   DATA[2577,13] := 828.5936;
   DATA[2577,14] := 1.0;
   DATA[2577,15] := 2.0;
   DATA[2577,16] := 1.0;
   DATA[2577,17] := 1.0;
   DATA[2577,18] := 1.0;
   DATA[2577,19] := 2.0;
   DATA[2577,20] := 148.808;
   DATA[2577,21] := 155.191;
   DATA[2577,22] := 1.713261;
   DATA[2577,23] := 874.6988;
   DATA[2577,24] := 2.0;
   DATA[2577,25] := 2.0;
   DATA[2577,26] := 7.871251;
   DATA[2577,27] := 144.4758;
   DATA[2577,28] := 261.3753;
   DATA[2577,29] := 12.03538;
   DATA[2577,30] := 1.724301;
   DATA[2577,31] := 1.29243;
   DATA[2577,32] := 0.7352687;
   DATA[2577,33] := 0.3084265;
   DATA[2577,34] := 2.0;
   DATA[2577,35] := 249.6155;
   DATA[2577,36] := 1.649953;
   DATA[2577,37] := 188.5254;
   DATA[2577,38] := 0.000128152;
   DATA[2577,39] := 1.0;
   DATA[2577,40] := 1.0;
   DATA[2578,0] := 2.550043;
   DATA[2578,1] := 868.9383;
   DATA[2578,2] := 2.0;
   DATA[2578,3] := 2.0;
   DATA[2578,4] := 262.3366;
   DATA[2578,5] := 8.396437;
   DATA[2578,6] := 329.4027;
   DATA[2578,7] := 2.452312;
   DATA[2578,8] := 2.0;
   DATA[2578,9] := 2.0;
   DATA[2578,10] := 2.0;
   DATA[2578,11] := 19.68756;
   DATA[2578,12] := 2.209653;
   DATA[2578,13] := 829.0342;
   DATA[2578,14] := 1.0;
   DATA[2578,15] := 2.0;
   DATA[2578,16] := 1.0;
   DATA[2578,17] := 1.0;
   DATA[2578,18] := 1.0;
   DATA[2578,19] := 2.0;
   DATA[2578,20] := 148.808;
   DATA[2578,21] := 155.191;
   DATA[2578,22] := 1.713261;
   DATA[2578,23] := 874.8141;
   DATA[2578,24] := 2.0;
   DATA[2578,25] := 2.0;
   DATA[2578,26] := 7.872853;
   DATA[2578,27] := 144.4758;
   DATA[2578,28] := 261.3753;
   DATA[2578,29] := 12.03538;
   DATA[2578,30] := 1.724301;
   DATA[2578,31] := 1.301524;
   DATA[2578,32] := 0.7352687;
   DATA[2578,33] := 0.3084265;
   DATA[2578,34] := 2.0;
   DATA[2578,35] := 249.8718;
   DATA[2578,36] := 1.649953;
   DATA[2578,37] := 188.7176;
   DATA[2578,38] := 0.000128152;
   DATA[2578,39] := 1.0;
   DATA[2578,40] := 1.0;
   DATA[2579,0] := 2.586875;
   DATA[2579,1] := 868.5458;
   DATA[2579,2] := 2.0;
   DATA[2579,3] := 2.0;
   DATA[2579,4] := 262.3366;
   DATA[2579,5] := 8.396437;
   DATA[2579,6] := 329.4027;
   DATA[2579,7] := 2.451927;
   DATA[2579,8] := 2.0;
   DATA[2579,9] := 2.0;
   DATA[2579,10] := 2.0;
   DATA[2579,11] := 19.71957;
   DATA[2579,12] := 2.209653;
   DATA[2579,13] := 829.3547;
   DATA[2579,14] := 1.0;
   DATA[2579,15] := 2.0;
   DATA[2579,16] := 1.0;
   DATA[2579,17] := 1.0;
   DATA[2579,18] := 1.0;
   DATA[2579,19] := 2.0;
   DATA[2579,20] := 148.808;
   DATA[2579,21] := 155.191;
   DATA[2579,22] := 1.716208;
   DATA[2579,23] := 875.0064;
   DATA[2579,24] := 2.0;
   DATA[2579,25] := 2.0;
   DATA[2579,26] := 7.872853;
   DATA[2579,27] := 144.4758;
   DATA[2579,28] := 261.3753;
   DATA[2579,29] := 12.03538;
   DATA[2579,30] := 1.724686;
   DATA[2579,31] := 1.296657;
   DATA[2579,32] := 0.7352687;
   DATA[2579,33] := 0.3084265;
   DATA[2579,34] := 2.0;
   DATA[2579,35] := 249.8718;
   DATA[2579,36] := 1.649953;
   DATA[2579,37] := 188.7176;
   DATA[2579,38] := 0.000128152;
   DATA[2579,39] := 1.0;
   DATA[2579,40] := 1.0;
   DATA[2580,0] := 2.632995;
   DATA[2580,1] := 868.5458;
   DATA[2580,2] := 2.0;
   DATA[2580,3] := 2.0;
   DATA[2580,4] := 262.3366;
   DATA[2580,5] := 8.396437;
   DATA[2580,6] := 329.4027;
   DATA[2580,7] := 2.451927;
   DATA[2580,8] := 2.0;
   DATA[2580,9] := 2.0;
   DATA[2580,10] := 2.0;
   DATA[2580,11] := 19.74198;
   DATA[2580,12] := 2.208116;
   DATA[2580,13] := 830.4762;
   DATA[2580,14] := 1.0;
   DATA[2580,15] := 2.0;
   DATA[2580,16] := 1.0;
   DATA[2580,17] := 1.0;
   DATA[2580,18] := 1.0;
   DATA[2580,19] := 2.0;
   DATA[2580,20] := 148.808;
   DATA[2580,21] := 155.191;
   DATA[2580,22] := 1.716208;
   DATA[2580,23] := 875.314;
   DATA[2580,24] := 2.0;
   DATA[2580,25] := 2.0;
   DATA[2580,26] := 7.872853;
   DATA[2580,27] := 144.4758;
   DATA[2580,28] := 261.3753;
   DATA[2580,29] := 12.03538;
   DATA[2580,30] := 1.725711;
   DATA[2580,31] := 1.298578;
   DATA[2580,32] := 0.7352687;
   DATA[2580,33] := 0.3084265;
   DATA[2580,34] := 2.0;
   DATA[2580,35] := 249.8718;
   DATA[2580,36] := 1.665972;
   DATA[2580,37] := 188.7176;
   DATA[2580,38] := 0.000128152;
   DATA[2580,39] := 1.0;
   DATA[2580,40] := 1.0;
   DATA[2581,0] := 2.65061;
   DATA[2581,1] := 868.5458;
   DATA[2581,2] := 2.0;
   DATA[2581,3] := 2.0;
   DATA[2581,4] := 262.3366;
   DATA[2581,5] := 8.396437;
   DATA[2581,6] := 329.4027;
   DATA[2581,7] := 2.451927;
   DATA[2581,8] := 2.0;
   DATA[2581,9] := 2.0;
   DATA[2581,10] := 2.0;
   DATA[2581,11] := 19.76439;
   DATA[2581,12] := 2.208116;
   DATA[2581,13] := 830.8767;
   DATA[2581,14] := 1.0;
   DATA[2581,15] := 2.0;
   DATA[2581,16] := 1.0;
   DATA[2581,17] := 1.0;
   DATA[2581,18] := 1.0;
   DATA[2581,19] := 2.0;
   DATA[2581,20] := 148.808;
   DATA[2581,21] := 155.191;
   DATA[2581,22] := 1.716208;
   DATA[2581,23] := 875.3909;
   DATA[2581,24] := 2.0;
   DATA[2581,25] := 2.0;
   DATA[2581,26] := 7.874776;
   DATA[2581,27] := 144.4758;
   DATA[2581,28] := 261.3753;
   DATA[2581,29] := 12.03538;
   DATA[2581,30] := 1.725711;
   DATA[2581,31] := 1.302165;
   DATA[2581,32] := 0.7352687;
   DATA[2581,33] := 0.3084265;
   DATA[2581,34] := 2.0;
   DATA[2581,35] := 249.8718;
   DATA[2581,36] := 1.665972;
   DATA[2581,37] := 188.7176;
   DATA[2581,38] := 0.000128152;
   DATA[2581,39] := 1.0;
   DATA[2581,40] := 1.0;
   DATA[2582,0] := 2.66246;
   DATA[2582,1] := 868.3495;
   DATA[2582,2] := 2.0;
   DATA[2582,3] := 2.0;
   DATA[2582,4] := 262.3366;
   DATA[2582,5] := 8.396437;
   DATA[2582,6] := 329.4027;
   DATA[2582,7] := 2.451927;
   DATA[2582,8] := 2.0;
   DATA[2582,9] := 2.0;
   DATA[2582,10] := 2.0;
   DATA[2582,11] := 19.77079;
   DATA[2582,12] := 2.208116;
   DATA[2582,13] := 831.1971;
   DATA[2582,14] := 1.0;
   DATA[2582,15] := 2.0;
   DATA[2582,16] := 1.0;
   DATA[2582,17] := 1.0;
   DATA[2582,18] := 1.0;
   DATA[2582,19] := 2.0;
   DATA[2582,20] := 148.808;
   DATA[2582,21] := 155.191;
   DATA[2582,22] := 1.716208;
   DATA[2582,23] := 875.3909;
   DATA[2582,24] := 2.0;
   DATA[2582,25] := 2.0;
   DATA[2582,26] := 7.874776;
   DATA[2582,27] := 144.4758;
   DATA[2582,28] := 261.3753;
   DATA[2582,29] := 12.03538;
   DATA[2582,30] := 1.725711;
   DATA[2582,31] := 1.296657;
   DATA[2582,32] := 0.7352687;
   DATA[2582,33] := 0.3084265;
   DATA[2582,34] := 2.0;
   DATA[2582,35] := 249.8718;
   DATA[2582,36] := 1.665972;
   DATA[2582,37] := 188.7176;
   DATA[2582,38] := 0.000128152;
   DATA[2582,39] := 1.0;
   DATA[2582,40] := 1.0;
   DATA[2583,0] := 2.666624;
   DATA[2583,1] := 868.4673;
   DATA[2583,2] := 2.0;
   DATA[2583,3] := 2.0;
   DATA[2583,4] := 262.3366;
   DATA[2583,5] := 8.396437;
   DATA[2583,6] := 329.4027;
   DATA[2583,7] := 2.451927;
   DATA[2583,8] := 2.0;
   DATA[2583,9] := 2.0;
   DATA[2583,10] := 2.0;
   DATA[2583,11] := 19.77079;
   DATA[2583,12] := 2.208116;
   DATA[2583,13] := 831.1971;
   DATA[2583,14] := 1.0;
   DATA[2583,15] := 2.0;
   DATA[2583,16] := 1.0;
   DATA[2583,17] := 1.0;
   DATA[2583,18] := 1.0;
   DATA[2583,19] := 2.0;
   DATA[2583,20] := 148.808;
   DATA[2583,21] := 155.3448;
   DATA[2583,22] := 1.716208;
   DATA[2583,23] := 876.0831;
   DATA[2583,24] := 2.0;
   DATA[2583,25] := 2.0;
   DATA[2583,26] := 7.874776;
   DATA[2583,27] := 144.4758;
   DATA[2583,28] := 261.3753;
   DATA[2583,29] := 12.03538;
   DATA[2583,30] := 1.725711;
   DATA[2583,31] := 1.291277;
   DATA[2583,32] := 0.7352687;
   DATA[2583,33] := 0.3084265;
   DATA[2583,34] := 2.0;
   DATA[2583,35] := 249.8718;
   DATA[2583,36] := 1.665972;
   DATA[2583,37] := 188.7176;
   DATA[2583,38] := 0.000128152;
   DATA[2583,39] := 1.0;
   DATA[2583,40] := 1.0;
   DATA[2584,0] := 2.63844;
   DATA[2584,1] := 868.114;
   DATA[2584,2] := 2.0;
   DATA[2584,3] := 2.0;
   DATA[2584,4] := 262.3366;
   DATA[2584,5] := 8.396437;
   DATA[2584,6] := 329.4027;
   DATA[2584,7] := 2.453209;
   DATA[2584,8] := 2.0;
   DATA[2584,9] := 2.0;
   DATA[2584,10] := 2.0;
   DATA[2584,11] := 19.71637;
   DATA[2584,12] := 2.208116;
   DATA[2584,13] := 831.3574;
   DATA[2584,14] := 1.0;
   DATA[2584,15] := 2.0;
   DATA[2584,16] := 1.0;
   DATA[2584,17] := 1.0;
   DATA[2584,18] := 1.0;
   DATA[2584,19] := 2.0;
   DATA[2584,20] := 148.808;
   DATA[2584,21] := 155.3448;
   DATA[2584,22] := 1.717746;
   DATA[2584,23] := 876.6983;
   DATA[2584,24] := 2.0;
   DATA[2584,25] := 2.0;
   DATA[2584,26] := 7.874776;
   DATA[2584,27] := 144.4758;
   DATA[2584,28] := 261.3753;
   DATA[2584,29] := 12.03538;
   DATA[2584,30] := 1.725711;
   DATA[2584,31] := 1.281286;
   DATA[2584,32] := 0.7352687;
   DATA[2584,33] := 0.3084265;
   DATA[2584,34] := 2.0;
   DATA[2584,35] := 249.9519;
   DATA[2584,36] := 1.665972;
   DATA[2584,37] := 188.7176;
   DATA[2584,38] := 0.000128152;
   DATA[2584,39] := 1.0;
   DATA[2584,40] := 1.0;
   DATA[2585,0] := 2.625308;
   DATA[2585,1] := 868.1533;
   DATA[2585,2] := 2.0;
   DATA[2585,3] := 2.0;
   DATA[2585,4] := 262.3366;
   DATA[2585,5] := 8.396437;
   DATA[2585,6] := 329.4027;
   DATA[2585,7] := 2.453849;
   DATA[2585,8] := 2.0;
   DATA[2585,9] := 2.0;
   DATA[2585,10] := 2.0;
   DATA[2585,11] := 19.68436;
   DATA[2585,12] := 2.208116;
   DATA[2585,13] := 831.1571;
   DATA[2585,14] := 1.0;
   DATA[2585,15] := 2.0;
   DATA[2585,16] := 1.0;
   DATA[2585,17] := 1.0;
   DATA[2585,18] := 1.0;
   DATA[2585,19] := 2.0;
   DATA[2585,20] := 148.808;
   DATA[2585,21] := 155.3448;
   DATA[2585,22] := 1.717746;
   DATA[2585,23] := 876.8521;
   DATA[2585,24] := 2.0;
   DATA[2585,25] := 2.0;
   DATA[2585,26] := 7.874776;
   DATA[2585,27] := 144.4758;
   DATA[2585,28] := 261.3753;
   DATA[2585,29] := 12.03538;
   DATA[2585,30] := 1.726737;
   DATA[2585,31] := 1.281286;
   DATA[2585,32] := 0.7352687;
   DATA[2585,33] := 0.3084265;
   DATA[2585,34] := 2.0;
   DATA[2585,35] := 250.016;
   DATA[2585,36] := 1.665972;
   DATA[2585,37] := 188.7176;
   DATA[2585,38] := 0.000128152;
   DATA[2585,39] := 1.0;
   DATA[2585,40] := 1.0;
   DATA[2586,0] := 2.611536;
   DATA[2586,1] := 867.7607;
   DATA[2586,2] := 2.0;
   DATA[2586,3] := 2.0;
   DATA[2586,4] := 262.3366;
   DATA[2586,5] := 8.396437;
   DATA[2586,6] := 329.4027;
   DATA[2586,7] := 2.455515;
   DATA[2586,8] := 2.0;
   DATA[2586,9] := 2.0;
   DATA[2586,10] := 2.0;
   DATA[2586,11] := 19.68436;
   DATA[2586,12] := 2.208116;
   DATA[2586,13] := 830.8367;
   DATA[2586,14] := 1.0;
   DATA[2586,15] := 2.0;
   DATA[2586,16] := 1.0;
   DATA[2586,17] := 1.0;
   DATA[2586,18] := 1.0;
   DATA[2586,19] := 2.0;
   DATA[2586,20] := 148.808;
   DATA[2586,21] := 155.3448;
   DATA[2586,22] := 1.714798;
   DATA[2586,23] := 877.1982;
   DATA[2586,24] := 2.0;
   DATA[2586,25] := 2.0;
   DATA[2586,26] := 7.874776;
   DATA[2586,27] := 144.4758;
   DATA[2586,28] := 261.3753;
   DATA[2586,29] := 12.03538;
   DATA[2586,30] := 1.726737;
   DATA[2586,31] := 1.288843;
   DATA[2586,32] := 0.7352687;
   DATA[2586,33] := 0.3084265;
   DATA[2586,34] := 2.0;
   DATA[2586,35] := 250.016;
   DATA[2586,36] := 1.665972;
   DATA[2586,37] := 188.8458;
   DATA[2586,38] := 0.000128152;
   DATA[2586,39] := 1.0;
   DATA[2586,40] := 1.0;
   DATA[2587,0] := 2.598725;
   DATA[2587,1] := 867.957;
   DATA[2587,2] := 2.0;
   DATA[2587,3] := 2.0;
   DATA[2587,4] := 262.3366;
   DATA[2587,5] := 8.396437;
   DATA[2587,6] := 329.4027;
   DATA[2587,7] := 2.455515;
   DATA[2587,8] := 2.0;
   DATA[2587,9] := 2.0;
   DATA[2587,10] := 2.0;
   DATA[2587,11] := 19.68436;
   DATA[2587,12] := 2.208116;
   DATA[2587,13] := 831.0369;
   DATA[2587,14] := 1.0;
   DATA[2587,15] := 2.0;
   DATA[2587,16] := 1.0;
   DATA[2587,17] := 1.0;
   DATA[2587,18] := 1.0;
   DATA[2587,19] := 2.0;
   DATA[2587,20] := 148.808;
   DATA[2587,21] := 155.2166;
   DATA[2587,22] := 1.714542;
   DATA[2587,23] := 877.4289;
   DATA[2587,24] := 2.0;
   DATA[2587,25] := 2.0;
   DATA[2587,26] := 7.874776;
   DATA[2587,27] := 144.4758;
   DATA[2587,28] := 261.3753;
   DATA[2587,29] := 12.03538;
   DATA[2587,30] := 1.725455;
   DATA[2587,31] := 1.281542;
   DATA[2587,32] := 0.7352687;
   DATA[2587,33] := 0.3084265;
   DATA[2587,34] := 2.0;
   DATA[2587,35] := 250.016;
   DATA[2587,36] := 1.665972;
   DATA[2587,37] := 188.8458;
   DATA[2587,38] := 0.000128152;
   DATA[2587,39] := 1.0;
   DATA[2587,40] := 1.0;
   DATA[2588,0] := 2.575665;
   DATA[2588,1] := 868.114;
   DATA[2588,2] := 2.0;
   DATA[2588,3] := 2.0;
   DATA[2588,4] := 262.3366;
   DATA[2588,5] := 8.395475;
   DATA[2588,6] := 329.4027;
   DATA[2588,7] := 2.455515;
   DATA[2588,8] := 2.0;
   DATA[2588,9] := 2.0;
   DATA[2588,10] := 2.0;
   DATA[2588,11] := 19.68436;
   DATA[2588,12] := 2.206963;
   DATA[2588,13] := 830.7966;
   DATA[2588,14] := 1.0;
   DATA[2588,15] := 2.0;
   DATA[2588,16] := 1.0;
   DATA[2588,17] := 1.0;
   DATA[2588,18] := 1.0;
   DATA[2588,19] := 2.0;
   DATA[2588,20] := 148.808;
   DATA[2588,21] := 155.2166;
   DATA[2588,22] := 1.714542;
   DATA[2588,23] := 877.3904;
   DATA[2588,24] := 2.0;
   DATA[2588,25] := 2.0;
   DATA[2588,26] := 7.874776;
   DATA[2588,27] := 144.4758;
   DATA[2588,28] := 261.3753;
   DATA[2588,29] := 12.03538;
   DATA[2588,30] := 1.725455;
   DATA[2588,31] := 1.271935;
   DATA[2588,32] := 0.7352687;
   DATA[2588,33] := 0.3084265;
   DATA[2588,34] := 2.0;
   DATA[2588,35] := 250.016;
   DATA[2588,36] := 1.665972;
   DATA[2588,37] := 188.8458;
   DATA[2588,38] := 0.000128152;
   DATA[2588,39] := 1.0;
   DATA[2588,40] := 1.0;
   DATA[2589,0] := 2.553886;
   DATA[2589,1] := 868.428;
   DATA[2589,2] := 2.0;
   DATA[2589,3] := 2.0;
   DATA[2589,4] := 262.3366;
   DATA[2589,5] := 8.395475;
   DATA[2589,6] := 329.4027;
   DATA[2589,7] := 2.455515;
   DATA[2589,8] := 2.0;
   DATA[2589,9] := 2.0;
   DATA[2589,10] := 2.0;
   DATA[2589,11] := 19.70357;
   DATA[2589,12] := 2.206707;
   DATA[2589,13] := 830.9568;
   DATA[2589,14] := 1.0;
   DATA[2589,15] := 2.0;
   DATA[2589,16] := 1.0;
   DATA[2589,17] := 1.0;
   DATA[2589,18] := 1.0;
   DATA[2589,19] := 2.0;
   DATA[2589,20] := 148.808;
   DATA[2589,21] := 155.2166;
   DATA[2589,22] := 1.714158;
   DATA[2589,23] := 877.5057;
   DATA[2589,24] := 2.0;
   DATA[2589,25] := 2.0;
   DATA[2589,26] := 7.874455;
   DATA[2589,27] := 144.4758;
   DATA[2589,28] := 261.3753;
   DATA[2589,29] := 12.03538;
   DATA[2589,30] := 1.725455;
   DATA[2589,31] := 1.270783;
   DATA[2589,32] := 0.7352687;
   DATA[2589,33] := 0.3084265;
   DATA[2589,34] := 2.0;
   DATA[2589,35] := 250.016;
   DATA[2589,36] := 1.665972;
   DATA[2589,37] := 188.8458;
   DATA[2589,38] := 0.000128152;
   DATA[2589,39] := 1.0;
   DATA[2589,40] := 1.0;
   DATA[2590,0] := 2.529225;
   DATA[2590,1] := 868.899;
   DATA[2590,2] := 2.0;
   DATA[2590,3] := 2.0;
   DATA[2590,4] := 262.3366;
   DATA[2590,5] := 8.395475;
   DATA[2590,6] := 329.4027;
   DATA[2590,7] := 2.454618;
   DATA[2590,8] := 2.0;
   DATA[2590,9] := 2.0;
   DATA[2590,10] := 2.0;
   DATA[2590,11] := 19.70357;
   DATA[2590,12] := 2.205554;
   DATA[2590,13] := 830.9969;
   DATA[2590,14] := 1.0;
   DATA[2590,15] := 2.0;
   DATA[2590,16] := 1.0;
   DATA[2590,17] := 1.0;
   DATA[2590,18] := 1.0;
   DATA[2590,19] := 2.0;
   DATA[2590,20] := 148.808;
   DATA[2590,21] := 155.2166;
   DATA[2590,22] := 1.713901;
   DATA[2590,23] := 877.5826;
   DATA[2590,24] := 2.0;
   DATA[2590,25] := 2.0;
   DATA[2590,26] := 7.873815;
   DATA[2590,27] := 144.4758;
   DATA[2590,28] := 261.3753;
   DATA[2590,29] := 12.03538;
   DATA[2590,30] := 1.726737;
   DATA[2590,31] := 1.279877;
   DATA[2590,32] := 0.7352687;
   DATA[2590,33] := 0.3084265;
   DATA[2590,34] := 2.0;
   DATA[2590,35] := 250.016;
   DATA[2590,36] := 1.665972;
   DATA[2590,37] := 188.8458;
   DATA[2590,38] := 0.000128152;
   DATA[2590,39] := 1.0;
   DATA[2590,40] := 1.0;
   DATA[2591,0] := 2.514493;
   DATA[2591,1] := 868.6635;
   DATA[2591,2] := 2.0;
   DATA[2591,3] := 2.0;
   DATA[2591,4] := 262.3366;
   DATA[2591,5] := 8.395475;
   DATA[2591,6] := 329.4027;
   DATA[2591,7] := 2.454618;
   DATA[2591,8] := 2.0;
   DATA[2591,9] := 2.0;
   DATA[2591,10] := 2.0;
   DATA[2591,11] := 19.76759;
   DATA[2591,12] := 2.204913;
   DATA[2591,13] := 830.8367;
   DATA[2591,14] := 1.0;
   DATA[2591,15] := 2.0;
   DATA[2591,16] := 1.0;
   DATA[2591,17] := 1.0;
   DATA[2591,18] := 1.0;
   DATA[2591,19] := 2.0;
   DATA[2591,20] := 148.808;
   DATA[2591,21] := 155.2166;
   DATA[2591,22] := 1.712876;
   DATA[2591,23] := 877.2366;
   DATA[2591,24] := 2.0;
   DATA[2591,25] := 2.0;
   DATA[2591,26] := 7.873815;
   DATA[2591,27] := 144.4758;
   DATA[2591,28] := 261.3753;
   DATA[2591,29] := 12.03538;
   DATA[2591,30] := 1.727506;
   DATA[2591,31] := 1.299731;
   DATA[2591,32] := 0.7352687;
   DATA[2591,33] := 0.3084265;
   DATA[2591,34] := 2.0;
   DATA[2591,35] := 250.016;
   DATA[2591,36] := 1.665972;
   DATA[2591,37] := 188.8458;
   DATA[2591,38] := 0.000128152;
   DATA[2591,39] := 1.0;
   DATA[2591,40] := 1.0;
   DATA[2592,0] := 2.493995;
   DATA[2592,1] := 868.8206;
   DATA[2592,2] := 2.0;
   DATA[2592,3] := 2.0;
   DATA[2592,4] := 262.3366;
   DATA[2592,5] := 8.395475;
   DATA[2592,6] := 329.4027;
   DATA[2592,7] := 2.453337;
   DATA[2592,8] := 2.0;
   DATA[2592,9] := 2.0;
   DATA[2592,10] := 2.0;
   DATA[2592,11] := 19.79;
   DATA[2592,12] := 2.204913;
   DATA[2592,13] := 831.1971;
   DATA[2592,14] := 1.0;
   DATA[2592,15] := 2.0;
   DATA[2592,16] := 1.0;
   DATA[2592,17] := 1.0;
   DATA[2592,18] := 1.0;
   DATA[2592,19] := 2.0;
   DATA[2592,20] := 148.808;
   DATA[2592,21] := 155.2166;
   DATA[2592,22] := 1.712876;
   DATA[2592,23] := 877.3904;
   DATA[2592,24] := 2.0;
   DATA[2592,25] := 2.0;
   DATA[2592,26] := 7.873815;
   DATA[2592,27] := 144.2707;
   DATA[2592,28] := 261.3753;
   DATA[2592,29] := 12.03538;
   DATA[2592,30] := 1.727506;
   DATA[2592,31] := 1.301524;
   DATA[2592,32] := 0.7352687;
   DATA[2592,33] := 0.3084265;
   DATA[2592,34] := 2.0;
   DATA[2592,35] := 250.016;
   DATA[2592,36] := 1.665972;
   DATA[2592,37] := 188.8458;
   DATA[2592,38] := 0.000128152;
   DATA[2592,39] := 1.0;
   DATA[2592,40] := 1.0;
   DATA[2593,0] := 2.480223;
   DATA[2593,1] := 868.6243;
   DATA[2593,2] := 2.0;
   DATA[2593,3] := 2.0;
   DATA[2593,4] := 262.3366;
   DATA[2593,5] := 8.395475;
   DATA[2593,6] := 329.4027;
   DATA[2593,7] := 2.453337;
   DATA[2593,8] := 2.0;
   DATA[2593,9] := 2.0;
   DATA[2593,10] := 2.0;
   DATA[2593,11] := 19.79;
   DATA[2593,12] := 2.204913;
   DATA[2593,13] := 830.6765;
   DATA[2593,14] := 1.0;
   DATA[2593,15] := 2.0;
   DATA[2593,16] := 1.0;
   DATA[2593,17] := 1.0;
   DATA[2593,18] := 1.0;
   DATA[2593,19] := 2.0;
   DATA[2593,20] := 148.808;
   DATA[2593,21] := 155.2166;
   DATA[2593,22] := 1.714926;
   DATA[2593,23] := 877.4673;
   DATA[2593,24] := 2.0;
   DATA[2593,25] := 2.0;
   DATA[2593,26] := 7.873815;
   DATA[2593,27] := 144.2707;
   DATA[2593,28] := 261.3753;
   DATA[2593,29] := 12.03538;
   DATA[2593,30] := 1.725455;
   DATA[2593,31] := 1.301652;
   DATA[2593,32] := 0.7352687;
   DATA[2593,33] := 0.3084265;
   DATA[2593,34] := 2.0;
   DATA[2593,35] := 250.016;
   DATA[2593,36] := 1.665972;
   DATA[2593,37] := 188.8458;
   DATA[2593,38] := 0.000128152;
   DATA[2593,39] := 1.0;
   DATA[2593,40] := 1.0;
   DATA[2594,0] := 2.452039;
   DATA[2594,1] := 868.6635;
   DATA[2594,2] := 2.0;
   DATA[2594,3] := 2.0;
   DATA[2594,4] := 262.3366;
   DATA[2594,5] := 8.395475;
   DATA[2594,6] := 329.4027;
   DATA[2594,7] := 2.453337;
   DATA[2594,8] := 2.0;
   DATA[2594,9] := 2.0;
   DATA[2594,10] := 2.0;
   DATA[2594,11] := 19.83482;
   DATA[2594,12] := 2.207091;
   DATA[2594,13] := 830.9969;
   DATA[2594,14] := 1.0;
   DATA[2594,15] := 2.0;
   DATA[2594,16] := 1.0;
   DATA[2594,17] := 1.0;
   DATA[2594,18] := 1.0;
   DATA[2594,19] := 2.0;
   DATA[2594,20] := 148.808;
   DATA[2594,21] := 155.2166;
   DATA[2594,22] := 1.716721;
   DATA[2594,23] := 877.1982;
   DATA[2594,24] := 2.0;
   DATA[2594,25] := 2.0;
   DATA[2594,26] := 7.873815;
   DATA[2594,27] := 144.2707;
   DATA[2594,28] := 261.4394;
   DATA[2594,29] := 12.03538;
   DATA[2594,30] := 1.725455;
   DATA[2594,31] := 1.292814;
   DATA[2594,32] := 0.7352687;
   DATA[2594,33] := 0.3084265;
   DATA[2594,34] := 2.0;
   DATA[2594,35] := 250.016;
   DATA[2594,36] := 1.665972;
   DATA[2594,37] := 188.8458;
   DATA[2594,38] := 0.000128152;
   DATA[2594,39] := 1.0;
   DATA[2594,40] := 1.0;
   DATA[2595,0] := 2.435384;
   DATA[2595,1] := 868.3495;
   DATA[2595,2] := 2.0;
   DATA[2595,3] := 2.0;
   DATA[2595,4] := 262.3366;
   DATA[2595,5] := 8.395475;
   DATA[2595,6] := 329.3258;
   DATA[2595,7] := 2.450774;
   DATA[2595,8] := 2.0;
   DATA[2595,9] := 2.0;
   DATA[2595,10] := 2.0;
   DATA[2595,11] := 19.85402;
   DATA[2595,12] := 2.207091;
   DATA[2595,13] := 830.7565;
   DATA[2595,14] := 1.0;
   DATA[2595,15] := 2.0;
   DATA[2595,16] := 1.0;
   DATA[2595,17] := 1.0;
   DATA[2595,18] := 1.0;
   DATA[2595,19] := 2.0;
   DATA[2595,20] := 148.808;
   DATA[2595,21] := 155.2166;
   DATA[2595,22] := 1.717874;
   DATA[2595,23] := 877.1982;
   DATA[2595,24] := 2.0;
   DATA[2595,25] := 2.0;
   DATA[2595,26] := 7.873815;
   DATA[2595,27] := 144.2707;
   DATA[2595,28] := 261.4394;
   DATA[2595,29] := 12.03538;
   DATA[2595,30] := 1.725455;
   DATA[2595,31] := 1.281927;
   DATA[2595,32] := 0.7352687;
   DATA[2595,33] := 0.3084265;
   DATA[2595,34] := 2.0;
   DATA[2595,35] := 250.016;
   DATA[2595,36] := 1.665972;
   DATA[2595,37] := 188.8458;
   DATA[2595,38] := 0.000128152;
   DATA[2595,39] := 1.0;
   DATA[2595,40] := 1.0;
   DATA[2596,0] := 2.435384;
   DATA[2596,1] := 868.3102;
   DATA[2596,2] := 2.0;
   DATA[2596,3] := 2.0;
   DATA[2596,4] := 262.3366;
   DATA[2596,5] := 8.395475;
   DATA[2596,6] := 329.3258;
   DATA[2596,7] := 2.450774;
   DATA[2596,8] := 2.0;
   DATA[2596,9] := 2.0;
   DATA[2596,10] := 2.0;
   DATA[2596,11] := 19.85402;
   DATA[2596,12] := 2.209525;
   DATA[2596,13] := 830.6765;
   DATA[2596,14] := 1.0;
   DATA[2596,15] := 2.0;
   DATA[2596,16] := 1.0;
   DATA[2596,17] := 1.0;
   DATA[2596,18] := 1.0;
   DATA[2596,19] := 2.0;
   DATA[2596,20] := 148.808;
   DATA[2596,21] := 155.2166;
   DATA[2596,22] := 1.717874;
   DATA[2596,23] := 877.1982;
   DATA[2596,24] := 2.0;
   DATA[2596,25] := 2.0;
   DATA[2596,26] := 7.873815;
   DATA[2596,27] := 144.2707;
   DATA[2596,28] := 261.5675;
   DATA[2596,29] := 12.03538;
   DATA[2596,30] := 1.725455;
   DATA[2596,31] := 1.288075;
   DATA[2596,32] := 0.7352687;
   DATA[2596,33] := 0.3084265;
   DATA[2596,34] := 2.0;
   DATA[2596,35] := 250.016;
   DATA[2596,36] := 1.665972;
   DATA[2596,37] := 188.8458;
   DATA[2596,38] := 0.000128152;
   DATA[2596,39] := 1.0;
   DATA[2596,40] := 1.0;
   DATA[2597,0] := 2.435064;
   DATA[2597,1] := 868.3102;
   DATA[2597,2] := 2.0;
   DATA[2597,3] := 2.0;
   DATA[2597,4] := 262.3366;
   DATA[2597,5] := 8.395475;
   DATA[2597,6] := 329.3258;
   DATA[2597,7] := 2.450774;
   DATA[2597,8] := 2.0;
   DATA[2597,9] := 2.0;
   DATA[2597,10] := 2.0;
   DATA[2597,11] := 19.7868;
   DATA[2597,12] := 2.209525;
   DATA[2597,13] := 830.3961;
   DATA[2597,14] := 1.0;
   DATA[2597,15] := 2.0;
   DATA[2597,16] := 1.0;
   DATA[2597,17] := 1.0;
   DATA[2597,18] := 1.0;
   DATA[2597,19] := 2.0;
   DATA[2597,20] := 148.808;
   DATA[2597,21] := 155.2166;
   DATA[2597,22] := 1.718771;
   DATA[2597,23] := 877.3904;
   DATA[2597,24] := 2.0;
   DATA[2597,25] := 2.0;
   DATA[2597,26] := 7.873815;
   DATA[2597,27] := 144.322;
   DATA[2597,28] := 261.5675;
   DATA[2597,29] := 12.03538;
   DATA[2597,30] := 1.725455;
   DATA[2597,31] := 1.286282;
   DATA[2597,32] := 0.7352687;
   DATA[2597,33] := 0.3069532;
   DATA[2597,34] := 2.0;
   DATA[2597,35] := 250.016;
   DATA[2597,36] := 1.665972;
   DATA[2597,37] := 188.8458;
   DATA[2597,38] := 0.000128152;
   DATA[2597,39] := 1.0;
   DATA[2597,40] := 1.0;
   DATA[2598,0] := 2.485667;
   DATA[2598,1] := 868.7421;
   DATA[2598,2] := 2.0;
   DATA[2598,3] := 2.0;
   DATA[2598,4] := 262.3366;
   DATA[2598,5] := 8.395475;
   DATA[2598,6] := 329.1464;
   DATA[2598,7] := 2.452055;
   DATA[2598,8] := 2.0;
   DATA[2598,9] := 2.0;
   DATA[2598,10] := 2.0;
   DATA[2598,11] := 19.7804;
   DATA[2598,12] := 2.209525;
   DATA[2598,13] := 830.5563;
   DATA[2598,14] := 1.0;
   DATA[2598,15] := 2.0;
   DATA[2598,16] := 1.0;
   DATA[2598,17] := 1.0;
   DATA[2598,18] := 1.0;
   DATA[2598,19] := 2.0;
   DATA[2598,20] := 148.808;
   DATA[2598,21] := 155.2166;
   DATA[2598,22] := 1.719284;
   DATA[2598,23] := 877.0828;
   DATA[2598,24] := 2.0;
   DATA[2598,25] := 2.0;
   DATA[2598,26] := 7.873815;
   DATA[2598,27] := 144.6039;
   DATA[2598,28] := 261.5675;
   DATA[2598,29] := 12.03538;
   DATA[2598,30] := 1.725455;
   DATA[2598,31] := 1.289228;
   DATA[2598,32] := 0.7352687;
   DATA[2598,33] := 0.306761;
   DATA[2598,34] := 2.0;
   DATA[2598,35] := 250.016;
   DATA[2598,36] := 1.665972;
   DATA[2598,37] := 188.8458;
   DATA[2598,38] := 0.000128152;
   DATA[2598,39] := 1.0;
   DATA[2598,40] := 1.0;
   DATA[2599,0] := 2.524421;
   DATA[2599,1] := 869.2523;
   DATA[2599,2] := 2.0;
   DATA[2599,3] := 2.0;
   DATA[2599,4] := 262.3366;
   DATA[2599,5] := 8.397718;
   DATA[2599,6] := 329.1464;
   DATA[2599,7] := 2.452055;
   DATA[2599,8] := 2.0;
   DATA[2599,9] := 2.0;
   DATA[2599,10] := 2.0;
   DATA[2599,11] := 19.75479;
   DATA[2599,12] := 2.209525;
   DATA[2599,13] := 830.5963;
   DATA[2599,14] := 1.0;
   DATA[2599,15] := 2.0;
   DATA[2599,16] := 1.0;
   DATA[2599,17] := 1.0;
   DATA[2599,18] := 1.0;
   DATA[2599,19] := 2.0;
   DATA[2599,20] := 148.808;
   DATA[2599,21] := 155.2166;
   DATA[2599,22] := 1.719284;
   DATA[2599,23] := 877.1213;
   DATA[2599,24] := 2.0;
   DATA[2599,25] := 2.0;
   DATA[2599,26] := 7.873815;
   DATA[2599,27] := 144.6039;
   DATA[2599,28] := 261.5675;
   DATA[2599,29] := 12.03538;
   DATA[2599,30] := 1.726865;
   DATA[2599,31] := 1.291918;
   DATA[2599,32] := 0.7352687;
   DATA[2599,33] := 0.3084265;
   DATA[2599,34] := 2.0;
   DATA[2599,35] := 250.2243;
   DATA[2599,36] := 1.665972;
   DATA[2599,37] := 189.006;
   DATA[2599,38] := 0.000128152;
   DATA[2599,39] := 1.0;
   DATA[2599,40] := 1.0;
   DATA[2600,0] := 2.562854;
   DATA[2600,1] := 869.8019;
   DATA[2600,2] := 2.0;
   DATA[2600,3] := 2.0;
   DATA[2600,4] := 262.3366;
   DATA[2600,5] := 8.397718;
   DATA[2600,6] := 329.1464;
   DATA[2600,7] := 2.452952;
   DATA[2600,8] := 2.0;
   DATA[2600,9] := 2.0;
   DATA[2600,10] := 2.0;
   DATA[2600,11] := 19.75479;
   DATA[2600,12] := 2.209525;
   DATA[2600,13] := 830.1958;
   DATA[2600,14] := 1.0;
   DATA[2600,15] := 2.0;
   DATA[2600,16] := 1.0;
   DATA[2600,17] := 1.0;
   DATA[2600,18] := 1.0;
   DATA[2600,19] := 2.0;
   DATA[2600,20] := 148.808;
   DATA[2600,21] := 155.2166;
   DATA[2600,22] := 1.719284;
   DATA[2600,23] := 877.3135;
   DATA[2600,24] := 2.0;
   DATA[2600,25] := 2.0;
   DATA[2600,26] := 7.873815;
   DATA[2600,27] := 144.5783;
   DATA[2600,28] := 261.5675;
   DATA[2600,29] := 12.03538;
   DATA[2600,30] := 1.72725;
   DATA[2600,31] := 1.282439;
   DATA[2600,32] := 0.7352687;
   DATA[2600,33] := 0.3084265;
   DATA[2600,34] := 2.0;
   DATA[2600,35] := 250.2243;
   DATA[2600,36] := 1.778105;
   DATA[2600,37] := 189.006;
   DATA[2600,38] := 0.000128152;
   DATA[2600,39] := 1.0;
   DATA[2600,40] := 1.0;
   DATA[2601,0] := 2.595522;
   DATA[2601,1] := 869.8019;
   DATA[2601,2] := 2.0;
   DATA[2601,3] := 2.0;
   DATA[2601,4] := 262.3366;
   DATA[2601,5] := 8.397718;
   DATA[2601,6] := 329.1464;
   DATA[2601,7] := 2.453593;
   DATA[2601,8] := 2.0;
   DATA[2601,9] := 2.0;
   DATA[2601,10] := 2.0;
   DATA[2601,11] := 19.75479;
   DATA[2601,12] := 2.205426;
   DATA[2601,13] := 830.5963;
   DATA[2601,14] := 1.0;
   DATA[2601,15] := 2.0;
   DATA[2601,16] := 1.0;
   DATA[2601,17] := 1.0;
   DATA[2601,18] := 1.0;
   DATA[2601,19] := 2.0;
   DATA[2601,20] := 148.808;
   DATA[2601,21] := 155.2166;
   DATA[2601,22] := 1.719284;
   DATA[2601,23] := 877.3904;
   DATA[2601,24] := 2.0;
   DATA[2601,25] := 2.0;
   DATA[2601,26] := 7.873815;
   DATA[2601,27] := 144.527;
   DATA[2601,28] := 261.5675;
   DATA[2601,29] := 12.03538;
   DATA[2601,30] := 1.72725;
   DATA[2601,31] := 1.281927;
   DATA[2601,32] := 0.7352687;
   DATA[2601,33] := 0.3084265;
   DATA[2601,34] := 2.0;
   DATA[2601,35] := 250.2243;
   DATA[2601,36] := 1.778105;
   DATA[2601,37] := 189.1983;
   DATA[2601,38] := 0.000128152;
   DATA[2601,39] := 1.0;
   DATA[2601,40] := 1.0;
   DATA[2602,0] := 2.628191;
   DATA[2602,1] := 869.2523;
   DATA[2602,2] := 2.0;
   DATA[2602,3] := 2.0;
   DATA[2602,4] := 262.3366;
   DATA[2602,5] := 8.397718;
   DATA[2602,6] := 329.1464;
   DATA[2602,7] := 2.453593;
   DATA[2602,8] := 2.0;
   DATA[2602,9] := 2.0;
   DATA[2602,10] := 2.0;
   DATA[2602,11] := 19.75479;
   DATA[2602,12] := 2.205426;
   DATA[2602,13] := 830.2759;
   DATA[2602,14] := 1.0;
   DATA[2602,15] := 2.0;
   DATA[2602,16] := 1.0;
   DATA[2602,17] := 1.0;
   DATA[2602,18] := 1.0;
   DATA[2602,19] := 2.0;
   DATA[2602,20] := 148.808;
   DATA[2602,21] := 155.3192;
   DATA[2602,22] := 1.719284;
   DATA[2602,23] := 877.3135;
   DATA[2602,24] := 2.0;
   DATA[2602,25] := 2.0;
   DATA[2602,26] := 7.873815;
   DATA[2602,27] := 144.5014;
   DATA[2602,28] := 261.5675;
   DATA[2602,29] := 12.03538;
   DATA[2602,30] := 1.72725;
   DATA[2602,31] := 1.277956;
   DATA[2602,32] := 0.7352687;
   DATA[2602,33] := 0.3084265;
   DATA[2602,34] := 2.0;
   DATA[2602,35] := 250.2243;
   DATA[2602,36] := 1.778105;
   DATA[2602,37] := 189.1983;
   DATA[2602,38] := 0.000128152;
   DATA[2602,39] := 1.0;
   DATA[2602,40] := 1.0;
   DATA[2603,0] := 2.64997;
   DATA[2603,1] := 869.5271;
   DATA[2603,2] := 2.0;
   DATA[2603,3] := 2.0;
   DATA[2603,4] := 262.3366;
   DATA[2603,5] := 8.397718;
   DATA[2603,6] := 329.1464;
   DATA[2603,7] := 2.453593;
   DATA[2603,8] := 2.0;
   DATA[2603,9] := 2.0;
   DATA[2603,10] := 2.0;
   DATA[2603,11] := 19.75479;
   DATA[2603,12] := 2.205426;
   DATA[2603,13] := 830.5963;
   DATA[2603,14] := 1.0;
   DATA[2603,15] := 2.0;
   DATA[2603,16] := 1.0;
   DATA[2603,17] := 1.0;
   DATA[2603,18] := 1.0;
   DATA[2603,19] := 2.0;
   DATA[2603,20] := 148.808;
   DATA[2603,21] := 155.3192;
   DATA[2603,22] := 1.719284;
   DATA[2603,23] := 877.4673;
   DATA[2603,24] := 2.0;
   DATA[2603,25] := 2.0;
   DATA[2603,26] := 7.873815;
   DATA[2603,27] := 144.5014;
   DATA[2603,28] := 261.5675;
   DATA[2603,29] := 12.03538;
   DATA[2603,30] := 1.72725;
   DATA[2603,31] := 1.272064;
   DATA[2603,32] := 0.7352687;
   DATA[2603,33] := 0.3084265;
   DATA[2603,34] := 2.0;
   DATA[2603,35] := 250.2243;
   DATA[2603,36] := 1.601897;
   DATA[2603,37] := 189.1983;
   DATA[2603,38] := 0.000128152;
   DATA[2603,39] := 1.0;
   DATA[2603,40] := 1.0;
   DATA[2604,0] := 2.660539;
   DATA[2604,1] := 869.6841;
   DATA[2604,2] := 2.0;
   DATA[2604,3] := 2.0;
   DATA[2604,4] := 262.3366;
   DATA[2604,5] := 8.397718;
   DATA[2604,6] := 329.3002;
   DATA[2604,7] := 2.453593;
   DATA[2604,8] := 2.0;
   DATA[2604,9] := 2.0;
   DATA[2604,10] := 2.0;
   DATA[2604,11] := 19.77399;
   DATA[2604,12] := 2.205426;
   DATA[2604,13] := 830.4762;
   DATA[2604,14] := 1.0;
   DATA[2604,15] := 2.0;
   DATA[2604,16] := 1.0;
   DATA[2604,17] := 1.0;
   DATA[2604,18] := 1.0;
   DATA[2604,19] := 2.0;
   DATA[2604,20] := 148.808;
   DATA[2604,21] := 155.3192;
   DATA[2604,22] := 1.719156;
   DATA[2604,23] := 877.8518;
   DATA[2604,24] := 2.0;
   DATA[2604,25] := 2.0;
   DATA[2604,26] := 7.873815;
   DATA[2604,27] := 144.3732;
   DATA[2604,28] := 261.4394;
   DATA[2604,29] := 12.03538;
   DATA[2604,30] := 1.72725;
   DATA[2604,31] := 1.281927;
   DATA[2604,32] := 0.7352687;
   DATA[2604,33] := 0.3081703;
   DATA[2604,34] := 2.0;
   DATA[2604,35] := 250.2403;
   DATA[2604,36] := 1.569859;
   DATA[2604,37] := 189.1983;
   DATA[2604,38] := 0.000128152;
   DATA[2604,39] := 1.0;
   DATA[2604,40] := 1.0;
   DATA[2605,0] := 2.649009;
   DATA[2605,1] := 869.8804;
   DATA[2605,2] := 2.0;
   DATA[2605,3] := 2.0;
   DATA[2605,4] := 262.3366;
   DATA[2605,5] := 8.397718;
   DATA[2605,6] := 329.3771;
   DATA[2605,7] := 2.452568;
   DATA[2605,8] := 2.0;
   DATA[2605,9] := 2.0;
   DATA[2605,10] := 2.0;
   DATA[2605,11] := 19.77399;
   DATA[2605,12] := 2.205426;
   DATA[2605,13] := 830.1958;
   DATA[2605,14] := 1.0;
   DATA[2605,15] := 2.0;
   DATA[2605,16] := 1.0;
   DATA[2605,17] := 1.0;
   DATA[2605,18] := 1.0;
   DATA[2605,19] := 2.0;
   DATA[2605,20] := 148.808;
   DATA[2605,21] := 155.473;
   DATA[2605,22] := 1.719156;
   DATA[2605,23] := 878.1594;
   DATA[2605,24] := 2.0;
   DATA[2605,25] := 2.0;
   DATA[2605,26] := 7.873815;
   DATA[2605,27] := 144.3732;
   DATA[2605,28] := 261.2471;
   DATA[2605,29] := 12.03538;
   DATA[2605,30] := 1.72725;
   DATA[2605,31] := 1.291533;
   DATA[2605,32] := 0.7352687;
   DATA[2605,33] := 0.3081703;
   DATA[2605,34] := 2.0;
   DATA[2605,35] := 250.3845;
   DATA[2605,36] := 1.569859;
   DATA[2605,37] := 189.1022;
   DATA[2605,38] := 0.000128152;
   DATA[2605,39] := 1.0;
   DATA[2605,40] := 1.0;
   DATA[2606,0] := 2.633956;
   DATA[2606,1] := 870.0374;
   DATA[2606,2] := 2.0;
   DATA[2606,3] := 2.0;
   DATA[2606,4] := 262.3366;
   DATA[2606,5] := 8.396757;
   DATA[2606,6] := 329.3771;
   DATA[2606,7] := 2.451415;
   DATA[2606,8] := 2.0;
   DATA[2606,9] := 2.0;
   DATA[2606,10] := 2.0;
   DATA[2606,11] := 19.72598;
   DATA[2606,12] := 2.205426;
   DATA[2606,13] := 830.0756;
   DATA[2606,14] := 1.0;
   DATA[2606,15] := 2.0;
   DATA[2606,16] := 1.0;
   DATA[2606,17] := 1.0;
   DATA[2606,18] := 1.0;
   DATA[2606,19] := 2.0;
   DATA[2606,20] := 148.808;
   DATA[2606,21] := 155.473;
   DATA[2606,22] := 1.719156;
   DATA[2606,23] := 877.9672;
   DATA[2606,24] := 2.0;
   DATA[2606,25] := 2.0;
   DATA[2606,26] := 7.873815;
   DATA[2606,27] := 144.3732;
   DATA[2606,28] := 261.2471;
   DATA[2606,29] := 12.03538;
   DATA[2606,30] := 1.72725;
   DATA[2606,31] := 1.292814;
   DATA[2606,32] := 0.7352687;
   DATA[2606,33] := 0.3081703;
   DATA[2606,34] := 2.0;
   DATA[2606,35] := 250.3845;
   DATA[2606,36] := 1.746067;
   DATA[2606,37] := 189.1022;
   DATA[2606,38] := 0.000128152;
   DATA[2606,39] := 1.0;
   DATA[2606,40] := 1.0;
   DATA[2607,0] := 2.616981;
   DATA[2607,1] := 870.2729;
   DATA[2607,2] := 2.0;
   DATA[2607,3] := 2.0;
   DATA[2607,4] := 262.3366;
   DATA[2607,5] := 8.394835;
   DATA[2607,6] := 329.3771;
   DATA[2607,7] := 2.451415;
   DATA[2607,8] := 2.0;
   DATA[2607,9] := 2.0;
   DATA[2607,10] := 2.0;
   DATA[2607,11] := 19.72598;
   DATA[2607,12] := 2.206194;
   DATA[2607,13] := 830.0356;
   DATA[2607,14] := 1.0;
   DATA[2607,15] := 2.0;
   DATA[2607,16] := 1.0;
   DATA[2607,17] := 1.0;
   DATA[2607,18] := 1.0;
   DATA[2607,19] := 2.0;
   DATA[2607,20] := 148.808;
   DATA[2607,21] := 155.473;
   DATA[2607,22] := 1.719156;
   DATA[2607,23] := 878.3517;
   DATA[2607,24] := 2.0;
   DATA[2607,25] := 2.0;
   DATA[2607,26] := 7.873815;
   DATA[2607,27] := 144.3732;
   DATA[2607,28] := 261.2471;
   DATA[2607,29] := 12.03538;
   DATA[2607,30] := 1.728147;
   DATA[2607,31] := 1.292814;
   DATA[2607,32] := 0.7352687;
   DATA[2607,33] := 0.3081703;
   DATA[2607,34] := 2.0;
   DATA[2607,35] := 250.3845;
   DATA[2607,36] := 1.746067;
   DATA[2607,37] := 189.1022;
   DATA[2607,38] := 0.000128152;
   DATA[2607,39] := 1.0;
   DATA[2607,40] := 1.0;
   DATA[2608,0] := 2.612177;
   DATA[2608,1] := 870.3121;
   DATA[2608,2] := 2.0;
   DATA[2608,3] := 2.0;
   DATA[2608,4] := 262.3366;
   DATA[2608,5] := 8.394835;
   DATA[2608,6] := 329.3771;
   DATA[2608,7] := 2.451415;
   DATA[2608,8] := 2.0;
   DATA[2608,9] := 2.0;
   DATA[2608,10] := 2.0;
   DATA[2608,11] := 19.72598;
   DATA[2608,12] := 2.206194;
   DATA[2608,13] := 829.7552;
   DATA[2608,14] := 1.0;
   DATA[2608,15] := 2.0;
   DATA[2608,16] := 1.0;
   DATA[2608,17] := 1.0;
   DATA[2608,18] := 1.0;
   DATA[2608,19] := 2.0;
   DATA[2608,20] := 148.808;
   DATA[2608,21] := 155.473;
   DATA[2608,22] := 1.720309;
   DATA[2608,23] := 878.2748;
   DATA[2608,24] := 2.0;
   DATA[2608,25] := 2.0;
   DATA[2608,26] := 7.873815;
   DATA[2608,27] := 144.3732;
   DATA[2608,28] := 261.2791;
   DATA[2608,29] := 12.03538;
   DATA[2608,30] := 1.728147;
   DATA[2608,31] := 1.300115;
   DATA[2608,32] := 0.7352687;
   DATA[2608,33] := 0.3081703;
   DATA[2608,34] := 2.0;
   DATA[2608,35] := 250.3845;
   DATA[2608,36] := 1.746067;
   DATA[2608,37] := 189.1022;
   DATA[2608,38] := 0.000128152;
   DATA[2608,39] := 1.0;
   DATA[2608,40] := 1.0;
   DATA[2609,0] := 2.600327;
   DATA[2609,1] := 870.2729;
   DATA[2609,2] := 2.0;
   DATA[2609,3] := 2.0;
   DATA[2609,4] := 262.3366;
   DATA[2609,5] := 8.394835;
   DATA[2609,6] := 329.3771;
   DATA[2609,7] := 2.450517;
   DATA[2609,8] := 2.0;
   DATA[2609,9] := 2.0;
   DATA[2609,10] := 2.0;
   DATA[2609,11] := 19.80601;
   DATA[2609,12] := 2.206194;
   DATA[2609,13] := 829.9555;
   DATA[2609,14] := 1.0;
   DATA[2609,15] := 2.0;
   DATA[2609,16] := 1.0;
   DATA[2609,17] := 1.0;
   DATA[2609,18] := 1.0;
   DATA[2609,19] := 2.0;
   DATA[2609,20] := 148.808;
   DATA[2609,21] := 155.473;
   DATA[2609,22] := 1.720437;
   DATA[2609,23] := 878.5824;
   DATA[2609,24] := 2.0;
   DATA[2609,25] := 2.0;
   DATA[2609,26] := 7.873815;
   DATA[2609,27] := 144.3732;
   DATA[2609,28] := 261.2791;
   DATA[2609,29] := 12.03538;
   DATA[2609,30] := 1.728147;
   DATA[2609,31] := 1.292046;
   DATA[2609,32] := 0.7352687;
   DATA[2609,33] := 0.3081703;
   DATA[2609,34] := 2.0;
   DATA[2609,35] := 250.3845;
   DATA[2609,36] := 1.746067;
   DATA[2609,37] := 189.1022;
   DATA[2609,38] := 0.000128152;
   DATA[2609,39] := 1.0;
   DATA[2609,40] := 1.0;
   DATA[2610,0] := 2.583352;
   DATA[2610,1] := 870.0767;
   DATA[2610,2] := 2.0;
   DATA[2610,3] := 2.0;
   DATA[2610,4] := 262.3366;
   DATA[2610,5] := 8.394835;
   DATA[2610,6] := 329.3771;
   DATA[2610,7] := 2.450517;
   DATA[2610,8] := 2.0;
   DATA[2610,9] := 2.0;
   DATA[2610,10] := 2.0;
   DATA[2610,11] := 19.80601;
   DATA[2610,12] := 2.206322;
   DATA[2610,13] := 829.8754;
   DATA[2610,14] := 1.0;
   DATA[2610,15] := 2.0;
   DATA[2610,16] := 1.0;
   DATA[2610,17] := 1.0;
   DATA[2610,18] := 1.0;
   DATA[2610,19] := 2.0;
   DATA[2610,20] := 148.808;
   DATA[2610,21] := 155.473;
   DATA[2610,22] := 1.720437;
   DATA[2610,23] := 878.1594;
   DATA[2610,24] := 2.0;
   DATA[2610,25] := 2.0;
   DATA[2610,26] := 7.873815;
   DATA[2610,27] := 144.3732;
   DATA[2610,28] := 261.2791;
   DATA[2610,29] := 12.03538;
   DATA[2610,30] := 1.730454;
   DATA[2610,31] := 1.292046;
   DATA[2610,32] := 0.7352687;
   DATA[2610,33] := 0.3084905;
   DATA[2610,34] := 2.0;
   DATA[2610,35] := 250.3845;
   DATA[2610,36] := 1.746067;
   DATA[2610,37] := 189.1823;
   DATA[2610,38] := 0.000128152;
   DATA[2610,39] := 1.0;
   DATA[2610,40] := 1.0;
   DATA[2611,0] := 2.553566;
   DATA[2611,1] := 870.3121;
   DATA[2611,2] := 2.0;
   DATA[2611,3] := 2.0;
   DATA[2611,4] := 262.3366;
   DATA[2611,5] := 8.394835;
   DATA[2611,6] := 329.3771;
   DATA[2611,7] := 2.450517;
   DATA[2611,8] := 2.0;
   DATA[2611,9] := 2.0;
   DATA[2611,10] := 2.0;
   DATA[2611,11] := 19.7804;
   DATA[2611,12] := 2.206835;
   DATA[2611,13] := 829.8353;
   DATA[2611,14] := 1.0;
   DATA[2611,15] := 2.0;
   DATA[2611,16] := 1.0;
   DATA[2611,17] := 1.0;
   DATA[2611,18] := 1.0;
   DATA[2611,19] := 2.0;
   DATA[2611,20] := 148.808;
   DATA[2611,21] := 155.473;
   DATA[2611,22] := 1.720437;
   DATA[2611,23] := 877.9672;
   DATA[2611,24] := 2.0;
   DATA[2611,25] := 2.0;
   DATA[2611,26] := 7.873815;
   DATA[2611,27] := 144.322;
   DATA[2611,28] := 261.4394;
   DATA[2611,29] := 12.03538;
   DATA[2611,30] := 1.730454;
   DATA[2611,31] := 1.297041;
   DATA[2611,32] := 0.7352687;
   DATA[2611,33] := 0.3084905;
   DATA[2611,34] := 2.0;
   DATA[2611,35] := 250.5608;
   DATA[2611,36] := 1.746067;
   DATA[2611,37] := 189.2624;
   DATA[2611,38] := 0.000128152;
   DATA[2611,39] := 1.0;
   DATA[2611,40] := 1.0;
   DATA[2612,0] := 2.535631;
   DATA[2612,1] := 870.5869;
   DATA[2612,2] := 2.0;
   DATA[2612,3] := 2.0;
   DATA[2612,4] := 262.3366;
   DATA[2612,5] := 8.394835;
   DATA[2612,6] := 329.3771;
   DATA[2612,7] := 2.450517;
   DATA[2612,8] := 2.0;
   DATA[2612,9] := 2.0;
   DATA[2612,10] := 2.0;
   DATA[2612,11] := 19.74198;
   DATA[2612,12] := 2.206835;
   DATA[2612,13] := 829.8754;
   DATA[2612,14] := 1.0;
   DATA[2612,15] := 2.0;
   DATA[2612,16] := 1.0;
   DATA[2612,17] := 1.0;
   DATA[2612,18] := 1.0;
   DATA[2612,19] := 2.0;
   DATA[2612,20] := 148.808;
   DATA[2612,21] := 155.473;
   DATA[2612,22] := 1.721334;
   DATA[2612,23] := 877.7749;
   DATA[2612,24] := 2.0;
   DATA[2612,25] := 2.0;
   DATA[2612,26] := 7.873815;
   DATA[2612,27] := 144.322;
   DATA[2612,28] := 261.4394;
   DATA[2612,29] := 12.03538;
   DATA[2612,30] := 1.730454;
   DATA[2612,31] := 1.283079;
   DATA[2612,32] := 0.7352687;
   DATA[2612,33] := 0.3084905;
   DATA[2612,34] := 2.0;
   DATA[2612,35] := 250.5608;
   DATA[2612,36] := 1.746067;
   DATA[2612,37] := 189.2624;
   DATA[2612,38] := 0.000128152;
   DATA[2612,39] := 1.0;
   DATA[2612,40] := 1.0;
   DATA[2613,0] := 2.513211;
   DATA[2613,1] := 870.3907;
   DATA[2613,2] := 2.0;
   DATA[2613,3] := 2.0;
   DATA[2613,4] := 262.3366;
   DATA[2613,5] := 8.394835;
   DATA[2613,6] := 329.3771;
   DATA[2613,7] := 2.451799;
   DATA[2613,8] := 2.0;
   DATA[2613,9] := 2.0;
   DATA[2613,10] := 2.0;
   DATA[2613,11] := 19.73878;
   DATA[2613,12] := 2.206835;
   DATA[2613,13] := 829.8754;
   DATA[2613,14] := 1.0;
   DATA[2613,15] := 2.0;
   DATA[2613,16] := 1.0;
   DATA[2613,17] := 1.0;
   DATA[2613,18] := 1.0;
   DATA[2613,19] := 2.0;
   DATA[2613,20] := 148.808;
   DATA[2613,21] := 155.3961;
   DATA[2613,22] := 1.721334;
   DATA[2613,23] := 878.0441;
   DATA[2613,24] := 2.0;
   DATA[2613,25] := 2.0;
   DATA[2613,26] := 7.873815;
   DATA[2613,27] := 144.322;
   DATA[2613,28] := 261.4394;
   DATA[2613,29] := 12.03538;
   DATA[2613,30] := 1.730454;
   DATA[2613,31] := 1.274881;
   DATA[2613,32] := 0.7352687;
   DATA[2613,33] := 0.3068251;
   DATA[2613,34] := 2.0;
   DATA[2613,35] := 250.3845;
   DATA[2613,36] := 1.746067;
   DATA[2613,37] := 189.2624;
   DATA[2613,38] := 0.000128152;
   DATA[2613,39] := 1.0;
   DATA[2613,40] := 1.0;
   DATA[2614,0] := 2.496877;
   DATA[2614,1] := 870.1944;
   DATA[2614,2] := 2.0;
   DATA[2614,3] := 2.0;
   DATA[2614,4] := 262.3366;
   DATA[2614,5] := 8.396757;
   DATA[2614,6] := 329.3771;
   DATA[2614,7] := 2.452696;
   DATA[2614,8] := 2.0;
   DATA[2614,9] := 2.0;
   DATA[2614,10] := 2.0;
   DATA[2614,11] := 19.70357;
   DATA[2614,12] := 2.206835;
   DATA[2614,13] := 830.1958;
   DATA[2614,14] := 1.0;
   DATA[2614,15] := 2.0;
   DATA[2614,16] := 1.0;
   DATA[2614,17] := 1.0;
   DATA[2614,18] := 1.0;
   DATA[2614,19] := 2.0;
   DATA[2614,20] := 148.808;
   DATA[2614,21] := 155.3961;
   DATA[2614,22] := 1.721334;
   DATA[2614,23] := 878.0441;
   DATA[2614,24] := 2.0;
   DATA[2614,25] := 2.0;
   DATA[2614,26] := 7.873815;
   DATA[2614,27] := 144.322;
   DATA[2614,28] := 261.4394;
   DATA[2614,29] := 12.03538;
   DATA[2614,30] := 1.730454;
   DATA[2614,31] := 1.26425;
   DATA[2614,32] := 0.7352687;
   DATA[2614,33] := 0.3068251;
   DATA[2614,34] := 2.0;
   DATA[2614,35] := 250.3845;
   DATA[2614,36] := 1.746067;
   DATA[2614,37] := 189.2624;
   DATA[2614,38] := 0.000128152;
   DATA[2614,39] := 1.0;
   DATA[2614,40] := 1.0;
   DATA[2615,0] := 2.469654;
   DATA[2615,1] := 870.0374;
   DATA[2615,2] := 2.0;
   DATA[2615,3] := 2.0;
   DATA[2615,4] := 262.3366;
   DATA[2615,5] := 8.396757;
   DATA[2615,6] := 329.2745;
   DATA[2615,7] := 2.452696;
   DATA[2615,8] := 2.0;
   DATA[2615,9] := 2.0;
   DATA[2615,10] := 2.0;
   DATA[2615,11] := 19.69396;
   DATA[2615,12] := 2.206835;
   DATA[2615,13] := 830.1958;
   DATA[2615,14] := 1.0;
   DATA[2615,15] := 2.0;
   DATA[2615,16] := 1.0;
   DATA[2615,17] := 1.0;
   DATA[2615,18] := 1.0;
   DATA[2615,19] := 2.0;
   DATA[2615,20] := 148.808;
   DATA[2615,21] := 155.3961;
   DATA[2615,22] := 1.719027;
   DATA[2615,23] := 877.8903;
   DATA[2615,24] := 2.0;
   DATA[2615,25] := 2.0;
   DATA[2615,26] := 7.873815;
   DATA[2615,27] := 144.322;
   DATA[2615,28] := 261.4394;
   DATA[2615,29] := 12.03538;
   DATA[2615,30] := 1.730454;
   DATA[2615,31] := 1.261432;
   DATA[2615,32] := 0.7352687;
   DATA[2615,33] := 0.3068251;
   DATA[2615,34] := 2.0;
   DATA[2615,35] := 250.2403;
   DATA[2615,36] := 1.746067;
   DATA[2615,37] := 189.0381;
   DATA[2615,38] := 0.000128152;
   DATA[2615,39] := 1.0;
   DATA[2615,40] := 1.0;
   DATA[2616,0] := 2.454601;
   DATA[2616,1] := 870.2729;
   DATA[2616,2] := 2.0;
   DATA[2616,3] := 2.0;
   DATA[2616,4] := 262.3366;
   DATA[2616,5] := 8.396757;
   DATA[2616,6] := 329.2745;
   DATA[2616,7] := 2.452696;
   DATA[2616,8] := 2.0;
   DATA[2616,9] := 2.0;
   DATA[2616,10] := 2.0;
   DATA[2616,11] := 19.77079;
   DATA[2616,12] := 2.206835;
   DATA[2616,13] := 830.4762;
   DATA[2616,14] := 1.0;
   DATA[2616,15] := 2.0;
   DATA[2616,16] := 1.0;
   DATA[2616,17] := 1.0;
   DATA[2616,18] := 1.0;
   DATA[2616,19] := 2.0;
   DATA[2616,20] := 148.808;
   DATA[2616,21] := 155.3961;
   DATA[2616,22] := 1.719027;
   DATA[2616,23] := 877.8134;
   DATA[2616,24] := 2.0;
   DATA[2616,25] := 2.0;
   DATA[2616,26] := 7.873815;
   DATA[2616,27] := 144.322;
   DATA[2616,28] := 261.4394;
   DATA[2616,29] := 12.03538;
   DATA[2616,30] := 1.729172;
   DATA[2616,31] := 1.261432;
   DATA[2616,32] := 0.7352687;
   DATA[2616,33] := 0.3068251;
   DATA[2616,34] := 2.0;
   DATA[2616,35] := 250.1602;
   DATA[2616,36] := 1.746067;
   DATA[2616,37] := 189.0381;
   DATA[2616,38] := 0.000128152;
   DATA[2616,39] := 1.0;
   DATA[2616,40] := 1.0;
   DATA[2617,0] := 2.435384;
   DATA[2617,1] := 870.0374;
   DATA[2617,2] := 2.0;
   DATA[2617,3] := 2.0;
   DATA[2617,4] := 262.3366;
   DATA[2617,5] := 8.396757;
   DATA[2617,6] := 329.2745;
   DATA[2617,7] := 2.452696;
   DATA[2617,8] := 2.0;
   DATA[2617,9] := 2.0;
   DATA[2617,10] := 2.0;
   DATA[2617,11] := 19.77079;
   DATA[2617,12] := 2.206835;
   DATA[2617,13] := 830.2358;
   DATA[2617,14] := 1.0;
   DATA[2617,15] := 2.0;
   DATA[2617,16] := 1.0;
   DATA[2617,17] := 1.0;
   DATA[2617,18] := 1.0;
   DATA[2617,19] := 2.0;
   DATA[2617,20] := 148.808;
   DATA[2617,21] := 155.3961;
   DATA[2617,22] := 1.717874;
   DATA[2617,23] := 877.698;
   DATA[2617,24] := 2.0;
   DATA[2617,25] := 2.0;
   DATA[2617,26] := 7.873815;
   DATA[2617,27] := 144.322;
   DATA[2617,28] := 261.4394;
   DATA[2617,29] := 12.03538;
   DATA[2617,30] := 1.729172;
   DATA[2617,31] := 1.272192;
   DATA[2617,32] := 0.7352687;
   DATA[2617,33] := 0.3068251;
   DATA[2617,34] := 2.0;
   DATA[2617,35] := 250.1602;
   DATA[2617,36] := 1.746067;
   DATA[2617,37] := 189.0381;
   DATA[2617,38] := 0.000128152;
   DATA[2617,39] := 1.0;
   DATA[2617,40] := 1.0;
   DATA[2618,0] := 2.428658;
   DATA[2618,1] := 869.4879;
   DATA[2618,2] := 2.0;
   DATA[2618,3] := 2.0;
   DATA[2618,4] := 262.3366;
   DATA[2618,5] := 8.396757;
   DATA[2618,6] := 329.2745;
   DATA[2618,7] := 2.452696;
   DATA[2618,8] := 2.0;
   DATA[2618,9] := 2.0;
   DATA[2618,10] := 2.0;
   DATA[2618,11] := 19.7836;
   DATA[2618,12] := 2.209909;
   DATA[2618,13] := 830.5563;
   DATA[2618,14] := 1.0;
   DATA[2618,15] := 2.0;
   DATA[2618,16] := 1.0;
   DATA[2618,17] := 1.0;
   DATA[2618,18] := 1.0;
   DATA[2618,19] := 2.0;
   DATA[2618,20] := 148.808;
   DATA[2618,21] := 155.3961;
   DATA[2618,22] := 1.717874;
   DATA[2618,23] := 877.8134;
   DATA[2618,24] := 2.0;
   DATA[2618,25] := 2.0;
   DATA[2618,26] := 7.873815;
   DATA[2618,27] := 144.322;
   DATA[2618,28] := 261.4394;
   DATA[2618,29] := 12.03538;
   DATA[2618,30] := 1.728147;
   DATA[2618,31] := 1.282823;
   DATA[2618,32] := 0.7352687;
   DATA[2618,33] := 0.3084265;
   DATA[2618,34] := 2.0;
   DATA[2618,35] := 250.1602;
   DATA[2618,36] := 1.746067;
   DATA[2618,37] := 189.0381;
   DATA[2618,38] := 0.000128152;
   DATA[2618,39] := 1.0;
   DATA[2618,40] := 1.0;
   DATA[2619,0] := 2.428338;
   DATA[2619,1] := 869.5271;
   DATA[2619,2] := 2.0;
   DATA[2619,3] := 2.0;
   DATA[2619,4] := 262.3366;
   DATA[2619,5] := 8.396757;
   DATA[2619,6] := 329.2745;
   DATA[2619,7] := 2.452696;
   DATA[2619,8] := 2.0;
   DATA[2619,9] := 2.0;
   DATA[2619,10] := 2.0;
   DATA[2619,11] := 19.82841;
   DATA[2619,12] := 2.209909;
   DATA[2619,13] := 830.9568;
   DATA[2619,14] := 1.0;
   DATA[2619,15] := 2.0;
   DATA[2619,16] := 1.0;
   DATA[2619,17] := 1.0;
   DATA[2619,18] := 1.0;
   DATA[2619,19] := 2.0;
   DATA[2619,20] := 148.808;
   DATA[2619,21] := 155.3961;
   DATA[2619,22] := 1.717874;
   DATA[2619,23] := 878.1979;
   DATA[2619,24] := 2.0;
   DATA[2619,25] := 2.0;
   DATA[2619,26] := 7.873815;
   DATA[2619,27] := 144.322;
   DATA[2619,28] := 261.4394;
   DATA[2619,29] := 12.03538;
   DATA[2619,30] := 1.726609;
   DATA[2619,31] := 1.300884;
   DATA[2619,32] := 0.7352687;
   DATA[2619,33] := 0.3084265;
   DATA[2619,34] := 2.0;
   DATA[2619,35] := 250.1602;
   DATA[2619,36] := 1.746067;
   DATA[2619,37] := 188.974;
   DATA[2619,38] := 0.000128152;
   DATA[2619,39] := 1.0;
   DATA[2619,40] := 1.0;
   DATA[2620,0] := 2.444352;
   DATA[2620,1] := 869.5271;
   DATA[2620,2] := 2.0;
   DATA[2620,3] := 2.0;
   DATA[2620,4] := 262.3366;
   DATA[2620,5] := 8.396757;
   DATA[2620,6] := 329.2745;
   DATA[2620,7] := 2.45449;
   DATA[2620,8] := 2.0;
   DATA[2620,9] := 2.0;
   DATA[2620,10] := 2.0;
   DATA[2620,11] := 19.82841;
   DATA[2620,12] := 2.209909;
   DATA[2620,13] := 831.1571;
   DATA[2620,14] := 1.0;
   DATA[2620,15] := 2.0;
   DATA[2620,16] := 1.0;
   DATA[2620,17] := 1.0;
   DATA[2620,18] := 1.0;
   DATA[2620,19] := 2.0;
   DATA[2620,20] := 148.808;
   DATA[2620,21] := 155.3961;
   DATA[2620,22] := 1.717874;
   DATA[2620,23] := 878.2363;
   DATA[2620,24] := 2.0;
   DATA[2620,25] := 2.0;
   DATA[2620,26] := 7.873815;
   DATA[2620,27] := 144.322;
   DATA[2620,28] := 261.4394;
   DATA[2620,29] := 12.03538;
   DATA[2620,30] := 1.726609;
   DATA[2620,31] := 1.302037;
   DATA[2620,32] := 0.7352687;
   DATA[2620,33] := 0.3084265;
   DATA[2620,34] := 2.0;
   DATA[2620,35] := 250.1602;
   DATA[2620,36] := 1.746067;
   DATA[2620,37] := 188.974;
   DATA[2620,38] := 0.000128152;
   DATA[2620,39] := 1.0;
   DATA[2620,40] := 1.0;
   DATA[2621,0] := 2.489831;
   DATA[2621,1] := 869.3308;
   DATA[2621,2] := 2.0;
   DATA[2621,3] := 2.0;
   DATA[2621,4] := 262.3366;
   DATA[2621,5] := 8.396757;
   DATA[2621,6] := 329.2745;
   DATA[2621,7] := 2.45449;
   DATA[2621,8] := 2.0;
   DATA[2621,9] := 2.0;
   DATA[2621,10] := 2.0;
   DATA[2621,11] := 19.76759;
   DATA[2621,12] := 2.212215;
   DATA[2621,13] := 831.077;
   DATA[2621,14] := 1.0;
   DATA[2621,15] := 2.0;
   DATA[2621,16] := 1.0;
   DATA[2621,17] := 1.0;
   DATA[2621,18] := 1.0;
   DATA[2621,19] := 2.0;
   DATA[2621,20] := 148.808;
   DATA[2621,21] := 155.3961;
   DATA[2621,22] := 1.717874;
   DATA[2621,23] := 878.2363;
   DATA[2621,24] := 2.0;
   DATA[2621,25] := 2.0;
   DATA[2621,26] := 7.873815;
   DATA[2621,27] := 144.4758;
   DATA[2621,28] := 261.3753;
   DATA[2621,29] := 12.03538;
   DATA[2621,30] := 1.726609;
   DATA[2621,31] := 1.310491;
   DATA[2621,32] := 0.7352687;
   DATA[2621,33] := 0.3084265;
   DATA[2621,34] := 2.0;
   DATA[2621,35] := 250.1602;
   DATA[2621,36] := 1.746067;
   DATA[2621,37] := 188.8939;
   DATA[2621,38] := 0.000128152;
   DATA[2621,39] := 1.0;
   DATA[2621,40] := 1.0;
   DATA[2622,0] := 2.528905;
   DATA[2622,1] := 869.2916;
   DATA[2622,2] := 2.0;
   DATA[2622,3] := 2.0;
   DATA[2622,4] := 262.3366;
   DATA[2622,5] := 8.396757;
   DATA[2622,6] := 329.2745;
   DATA[2622,7] := 2.45449;
   DATA[2622,8] := 2.0;
   DATA[2622,9] := 2.0;
   DATA[2622,10] := 2.0;
   DATA[2622,11] := 19.71957;
   DATA[2622,12] := 2.212728;
   DATA[2622,13] := 831.1971;
   DATA[2622,14] := 1.0;
   DATA[2622,15] := 2.0;
   DATA[2622,16] := 1.0;
   DATA[2622,17] := 1.0;
   DATA[2622,18] := 1.0;
   DATA[2622,19] := 2.0;
   DATA[2622,20] := 148.808;
   DATA[2622,21] := 155.3961;
   DATA[2622,22] := 1.717874;
   DATA[2622,23] := 878.0441;
   DATA[2622,24] := 2.0;
   DATA[2622,25] := 2.0;
   DATA[2622,26] := 7.873815;
   DATA[2622,27] := 144.4758;
   DATA[2622,28] := 261.3753;
   DATA[2622,29] := 12.03538;
   DATA[2622,30] := 1.726609;
   DATA[2622,31] := 1.311387;
   DATA[2622,32] := 0.7352687;
   DATA[2622,33] := 0.3084265;
   DATA[2622,34] := 2.0;
   DATA[2622,35] := 250.1602;
   DATA[2622,36] := 1.746067;
   DATA[2622,37] := 188.8779;
   DATA[2622,38] := 0.000128152;
   DATA[2622,39] := 1.0;
   DATA[2622,40] := 1.0;
   DATA[2623,0] := 2.571182;
   DATA[2623,1] := 869.2131;
   DATA[2623,2] := 2.0;
   DATA[2623,3] := 2.0;
   DATA[2623,4] := 262.3366;
   DATA[2623,5] := 8.396757;
   DATA[2623,6] := 329.2745;
   DATA[2623,7] := 2.45449;
   DATA[2623,8] := 2.0;
   DATA[2623,9] := 2.0;
   DATA[2623,10] := 2.0;
   DATA[2623,11] := 19.67796;
   DATA[2623,12] := 2.212728;
   DATA[2623,13] := 831.6778;
   DATA[2623,14] := 1.0;
   DATA[2623,15] := 2.0;
   DATA[2623,16] := 1.0;
   DATA[2623,17] := 1.0;
   DATA[2623,18] := 1.0;
   DATA[2623,19] := 2.0;
   DATA[2623,20] := 148.808;
   DATA[2623,21] := 155.3961;
   DATA[2623,22] := 1.715952;
   DATA[2623,23] := 878.1594;
   DATA[2623,24] := 2.0;
   DATA[2623,25] := 2.0;
   DATA[2623,26] := 7.873815;
   DATA[2623,27] := 144.4758;
   DATA[2623,28] := 261.3753;
   DATA[2623,29] := 12.03538;
   DATA[2623,30] := 1.726609;
   DATA[2623,31] := 1.302165;
   DATA[2623,32] := 0.7352687;
   DATA[2623,33] := 0.3068251;
   DATA[2623,34] := 2.0;
   DATA[2623,35] := 250.1602;
   DATA[2623,36] := 1.746067;
   DATA[2623,37] := 188.8779;
   DATA[2623,38] := 0.000128152;
   DATA[2623,39] := 1.0;
   DATA[2623,40] := 1.0;
   DATA[2624,0] := 2.603529;
   DATA[2624,1] := 869.2523;
   DATA[2624,2] := 2.0;
   DATA[2624,3] := 2.0;
   DATA[2624,4] := 262.3366;
   DATA[2624,5] := 8.396757;
   DATA[2624,6] := 329.2745;
   DATA[2624,7] := 2.45449;
   DATA[2624,8] := 2.0;
   DATA[2624,9] := 2.0;
   DATA[2624,10] := 2.0;
   DATA[2624,11] := 19.65235;
   DATA[2624,12] := 2.212215;
   DATA[2624,13] := 831.6778;
   DATA[2624,14] := 1.0;
   DATA[2624,15] := 2.0;
   DATA[2624,16] := 1.0;
   DATA[2624,17] := 1.0;
   DATA[2624,18] := 1.0;
   DATA[2624,19] := 2.0;
   DATA[2624,20] := 148.808;
   DATA[2624,21] := 155.3961;
   DATA[2624,22] := 1.715183;
   DATA[2624,23] := 878.3517;
   DATA[2624,24] := 2.0;
   DATA[2624,25] := 2.0;
   DATA[2624,26] := 7.873815;
   DATA[2624,27] := 144.4758;
   DATA[2624,28] := 261.3753;
   DATA[2624,29] := 12.03538;
   DATA[2624,30] := 1.725327;
   DATA[2624,31] := 1.30178;
   DATA[2624,32] := 0.7352687;
   DATA[2624,33] := 0.3068251;
   DATA[2624,34] := 2.0;
   DATA[2624,35] := 250.1602;
   DATA[2624,36] := 1.746067;
   DATA[2624,37] := 188.8779;
   DATA[2624,38] := 0.000128152;
   DATA[2624,39] := 1.0;
   DATA[2624,40] := 1.0;
   DATA[2625,0] := 2.63876;
   DATA[2625,1] := 868.9383;
   DATA[2625,2] := 2.0;
   DATA[2625,3] := 2.0;
   DATA[2625,4] := 262.3366;
   DATA[2625,5] := 8.396757;
   DATA[2625,6] := 329.2745;
   DATA[2625,7] := 2.456156;
   DATA[2625,8] := 2.0;
   DATA[2625,9] := 2.0;
   DATA[2625,10] := 2.0;
   DATA[2625,11] := 19.60753;
   DATA[2625,12] := 2.210678;
   DATA[2625,13] := 831.798;
   DATA[2625,14] := 1.0;
   DATA[2625,15] := 2.0;
   DATA[2625,16] := 1.0;
   DATA[2625,17] := 1.0;
   DATA[2625,18] := 1.0;
   DATA[2625,19] := 2.0;
   DATA[2625,20] := 148.808;
   DATA[2625,21] := 155.3961;
   DATA[2625,22] := 1.715183;
   DATA[2625,23] := 878.6208;
   DATA[2625,24] := 2.0;
   DATA[2625,25] := 2.0;
   DATA[2625,26] := 7.873815;
   DATA[2625,27] := 144.4758;
   DATA[2625,28] := 261.3753;
   DATA[2625,29] := 12.03538;
   DATA[2625,30] := 1.725327;
   DATA[2625,31] := 1.30178;
   DATA[2625,32] := 0.7352687;
   DATA[2625,33] := 0.3068251;
   DATA[2625,34] := 2.0;
   DATA[2625,35] := 250.1602;
   DATA[2625,36] := 1.665972;
   DATA[2625,37] := 188.8779;
   DATA[2625,38] := 0.000128152;
   DATA[2625,39] := 1.0;
   DATA[2625,40] := 1.0;
   DATA[2626,0] := 2.63876;
   DATA[2626,1] := 868.9383;
   DATA[2626,2] := 2.0;
   DATA[2626,3] := 2.0;
   DATA[2626,4] := 262.3366;
   DATA[2626,5] := 8.396757;
   DATA[2626,6] := 329.2745;
   DATA[2626,7] := 2.456156;
   DATA[2626,8] := 2.0;
   DATA[2626,9] := 2.0;
   DATA[2626,10] := 2.0;
   DATA[2626,11] := 19.60753;
   DATA[2626,12] := 2.210678;
   DATA[2626,13] := 831.798;
   DATA[2626,14] := 1.0;
   DATA[2626,15] := 2.0;
   DATA[2626,16] := 1.0;
   DATA[2626,17] := 1.0;
   DATA[2626,18] := 1.0;
   DATA[2626,19] := 2.0;
   DATA[2626,20] := 148.808;
   DATA[2626,21] := 155.3961;
   DATA[2626,22] := 1.715183;
   DATA[2626,23] := 878.6208;
   DATA[2626,24] := 2.0;
   DATA[2626,25] := 2.0;
   DATA[2626,26] := 7.873815;
   DATA[2626,27] := 144.4758;
   DATA[2626,28] := 261.3753;
   DATA[2626,29] := 12.03538;
   DATA[2626,30] := 1.725327;
   DATA[2626,31] := 1.30178;
   DATA[2626,32] := 0.7352687;
   DATA[2626,33] := 0.3068251;
   DATA[2626,34] := 2.0;
   DATA[2626,35] := 250.1602;
   DATA[2626,36] := 1.665972;
   DATA[2626,37] := 188.8779;
   DATA[2626,38] := 0.000128152;
   DATA[2626,39] := 1.0;
   DATA[2626,40] := 1.0;
   DATA[2627,0] := 2.653172;
   DATA[2627,1] := 869.4094;
   DATA[2627,2] := 2.0;
   DATA[2627,3] := 2.0;
   DATA[2627,4] := 262.3366;
   DATA[2627,5] := 8.396757;
   DATA[2627,6] := 329.2745;
   DATA[2627,7] := 2.456156;
   DATA[2627,8] := 2.0;
   DATA[2627,9] := 2.0;
   DATA[2627,10] := 2.0;
   DATA[2627,11] := 19.60753;
   DATA[2627,12] := 2.209269;
   DATA[2627,13] := 832.1584;
   DATA[2627,14] := 1.0;
   DATA[2627,15] := 2.0;
   DATA[2627,16] := 1.0;
   DATA[2627,17] := 1.0;
   DATA[2627,18] := 1.0;
   DATA[2627,19] := 2.0;
   DATA[2627,20] := 148.808;
   DATA[2627,21] := 155.3961;
   DATA[2627,22] := 1.716849;
   DATA[2627,23] := 878.7362;
   DATA[2627,24] := 2.0;
   DATA[2627,25] := 2.0;
   DATA[2627,26] := 7.873815;
   DATA[2627,27] := 144.4758;
   DATA[2627,28] := 261.3753;
   DATA[2627,29] := 12.03538;
   DATA[2627,30] := 1.725327;
   DATA[2627,31] := 1.30178;
   DATA[2627,32] := 0.7352687;
   DATA[2627,33] := 0.3068251;
   DATA[2627,34] := 2.0;
   DATA[2627,35] := 250.1602;
   DATA[2627,36] := 1.665972;
   DATA[2627,37] := 188.8779;
   DATA[2627,38] := 0.000128152;
   DATA[2627,39] := 1.0;
   DATA[2627,40] := 1.0;
   DATA[2628,0] := 2.654774;
   DATA[2628,1] := 869.0953;
   DATA[2628,2] := 2.0;
   DATA[2628,3] := 2.0;
   DATA[2628,4] := 262.3366;
   DATA[2628,5] := 8.396757;
   DATA[2628,6] := 329.2745;
   DATA[2628,7] := 2.456156;
   DATA[2628,8] := 2.0;
   DATA[2628,9] := 2.0;
   DATA[2628,10] := 2.0;
   DATA[2628,11] := 19.60753;
   DATA[2628,12] := 2.209269;
   DATA[2628,13] := 832.0383;
   DATA[2628,14] := 1.0;
   DATA[2628,15] := 2.0;
   DATA[2628,16] := 1.0;
   DATA[2628,17] := 1.0;
   DATA[2628,18] := 1.0;
   DATA[2628,19] := 2.0;
   DATA[2628,20] := 148.808;
   DATA[2628,21] := 155.5499;
   DATA[2628,22] := 1.718771;
   DATA[2628,23] := 878.5439;
   DATA[2628,24] := 2.0;
   DATA[2628,25] := 2.0;
   DATA[2628,26] := 7.873815;
   DATA[2628,27] := 144.4758;
   DATA[2628,28] := 261.3753;
   DATA[2628,29] := 12.03538;
   DATA[2628,30] := 1.725327;
   DATA[2628,31] := 1.294095;
   DATA[2628,32] := 0.7352687;
   DATA[2628,33] := 0.3068251;
   DATA[2628,34] := 2.0;
   DATA[2628,35] := 250.1602;
   DATA[2628,36] := 1.730048;
   DATA[2628,37] := 188.9419;
   DATA[2628,38] := 0.000128152;
   DATA[2628,39] := 1.0;
   DATA[2628,40] := 1.0;
   DATA[2629,0] := 2.636198;
   DATA[2629,1] := 869.2523;
   DATA[2629,2] := 2.0;
   DATA[2629,3] := 2.0;
   DATA[2629,4] := 262.3366;
   DATA[2629,5] := 8.396757;
   DATA[2629,6] := 329.2745;
   DATA[2629,7] := 2.456156;
   DATA[2629,8] := 2.0;
   DATA[2629,9] := 2.0;
   DATA[2629,10] := 2.0;
   DATA[2629,11] := 19.60753;
   DATA[2629,12] := 2.209269;
   DATA[2629,13] := 831.9582;
   DATA[2629,14] := 1.0;
   DATA[2629,15] := 2.0;
   DATA[2629,16] := 1.0;
   DATA[2629,17] := 1.0;
   DATA[2629,18] := 1.0;
   DATA[2629,19] := 2.0;
   DATA[2629,20] := 148.808;
   DATA[2629,21] := 155.5499;
   DATA[2629,22] := 1.72095;
   DATA[2629,23] := 878.6208;
   DATA[2629,24] := 2.0;
   DATA[2629,25] := 2.0;
   DATA[2629,26] := 7.873815;
   DATA[2629,27] := 144.4758;
   DATA[2629,28] := 261.3753;
   DATA[2629,29] := 12.03538;
   DATA[2629,30] := 1.72725;
   DATA[2629,31] := 1.291149;
   DATA[2629,32] := 0.7352687;
   DATA[2629,33] := 0.3068251;
   DATA[2629,34] := 2.0;
   DATA[2629,35] := 250.1602;
   DATA[2629,36] := 1.778105;
   DATA[2629,37] := 189.0861;
   DATA[2629,38] := 0.000128152;
   DATA[2629,39] := 1.0;
   DATA[2629,40] := 1.0;
   DATA[2630,0] := 2.622105;
   DATA[2630,1] := 868.7421;
   DATA[2630,2] := 2.0;
   DATA[2630,3] := 2.0;
   DATA[2630,4] := 262.3366;
   DATA[2630,5] := 8.396757;
   DATA[2630,6] := 329.2745;
   DATA[2630,7] := 2.456156;
   DATA[2630,8] := 2.0;
   DATA[2630,9] := 2.0;
   DATA[2630,10] := 2.0;
   DATA[2630,11] := 19.62994;
   DATA[2630,12] := 2.209269;
   DATA[2630,13] := 832.1584;
   DATA[2630,14] := 1.0;
   DATA[2630,15] := 2.0;
   DATA[2630,16] := 1.0;
   DATA[2630,17] := 1.0;
   DATA[2630,18] := 1.0;
   DATA[2630,19] := 2.0;
   DATA[2630,20] := 148.808;
   DATA[2630,21] := 155.5499;
   DATA[2630,22] := 1.72095;
   DATA[2630,23] := 878.1979;
   DATA[2630,24] := 2.0;
   DATA[2630,25] := 2.0;
   DATA[2630,26] := 7.873815;
   DATA[2630,27] := 144.4758;
   DATA[2630,28] := 261.3753;
   DATA[2630,29] := 12.03538;
   DATA[2630,30] := 1.728531;
   DATA[2630,31] := 1.282439;
   DATA[2630,32] := 0.7352687;
   DATA[2630,33] := 0.3080421;
   DATA[2630,34] := 2.0;
   DATA[2630,35] := 250.3044;
   DATA[2630,36] := 1.778105;
   DATA[2630,37] := 189.1823;
   DATA[2630,38] := 0.000128152;
   DATA[2630,39] := 1.0;
   DATA[2630,40] := 1.0;
   DATA[2631,0] := 2.6157;
   DATA[2631,1] := 869.1346;
   DATA[2631,2] := 2.0;
   DATA[2631,3] := 2.0;
   DATA[2631,4] := 262.3366;
   DATA[2631,5] := 8.396757;
   DATA[2631,6] := 329.2745;
   DATA[2631,7] := 2.456156;
   DATA[2631,8] := 2.0;
   DATA[2631,9] := 2.0;
   DATA[2631,10] := 2.0;
   DATA[2631,11] := 19.68756;
   DATA[2631,12] := 2.209269;
   DATA[2631,13] := 831.798;
   DATA[2631,14] := 1.0;
   DATA[2631,15] := 2.0;
   DATA[2631,16] := 1.0;
   DATA[2631,17] := 1.0;
   DATA[2631,18] := 1.0;
   DATA[2631,19] := 2.0;
   DATA[2631,20] := 148.808;
   DATA[2631,21] := 155.5499;
   DATA[2631,22] := 1.718771;
   DATA[2631,23] := 878.3901;
   DATA[2631,24] := 2.0;
   DATA[2631,25] := 2.0;
   DATA[2631,26] := 7.873815;
   DATA[2631,27] := 144.4758;
   DATA[2631,28] := 261.3753;
   DATA[2631,29] := 12.03538;
   DATA[2631,30] := 1.728531;
   DATA[2631,31] := 1.285129;
   DATA[2631,32] := 0.7352687;
   DATA[2631,33] := 0.3083624;
   DATA[2631,34] := 2.0;
   DATA[2631,35] := 250.3365;
   DATA[2631,36] := 1.778105;
   DATA[2631,37] := 189.1823;
   DATA[2631,38] := 0.000128152;
   DATA[2631,39] := 1.0;
   DATA[2631,40] := 1.0;
   DATA[2632,0] := 2.603209;
   DATA[2632,1] := 868.8206;
   DATA[2632,2] := 2.0;
   DATA[2632,3] := 2.0;
   DATA[2632,4] := 262.3366;
   DATA[2632,5] := 8.39868;
   DATA[2632,6] := 329.2745;
   DATA[2632,7] := 2.456156;
   DATA[2632,8] := 2.0;
   DATA[2632,9] := 2.0;
   DATA[2632,10] := 2.0;
   DATA[2632,11] := 19.69076;
   DATA[2632,12] := 2.207475;
   DATA[2632,13] := 832.0783;
   DATA[2632,14] := 1.0;
   DATA[2632,15] := 2.0;
   DATA[2632,16] := 1.0;
   DATA[2632,17] := 1.0;
   DATA[2632,18] := 1.0;
   DATA[2632,19] := 2.0;
   DATA[2632,20] := 148.808;
   DATA[2632,21] := 155.5499;
   DATA[2632,22] := 1.718771;
   DATA[2632,23] := 878.3517;
   DATA[2632,24] := 2.0;
   DATA[2632,25] := 2.0;
   DATA[2632,26] := 7.873815;
   DATA[2632,27] := 144.4758;
   DATA[2632,28] := 261.3753;
   DATA[2632,29] := 12.03538;
   DATA[2632,30] := 1.728531;
   DATA[2632,31] := 1.291405;
   DATA[2632,32] := 0.7352687;
   DATA[2632,33] := 0.3083624;
   DATA[2632,34] := 2.0;
   DATA[2632,35] := 250.4326;
   DATA[2632,36] := 1.778105;
   DATA[2632,37] := 189.1823;
   DATA[2632,38] := 0.000128152;
   DATA[2632,39] := 1.0;
   DATA[2632,40] := 1.0;
   DATA[2633,0] := 2.591359;
   DATA[2633,1] := 868.8598;
   DATA[2633,2] := 2.0;
   DATA[2633,3] := 2.0;
   DATA[2633,4] := 262.3366;
   DATA[2633,5] := 8.39868;
   DATA[2633,6] := 329.2745;
   DATA[2633,7] := 2.456156;
   DATA[2633,8] := 2.0;
   DATA[2633,9] := 2.0;
   DATA[2633,10] := 2.0;
   DATA[2633,11] := 19.71957;
   DATA[2633,12] := 2.206707;
   DATA[2633,13] := 832.0783;
   DATA[2633,14] := 1.0;
   DATA[2633,15] := 2.0;
   DATA[2633,16] := 1.0;
   DATA[2633,17] := 1.0;
   DATA[2633,18] := 1.0;
   DATA[2633,19] := 2.0;
   DATA[2633,20] := 148.808;
   DATA[2633,21] := 155.5499;
   DATA[2633,22] := 1.722359;
   DATA[2633,23] := 878.3901;
   DATA[2633,24] := 2.0;
   DATA[2633,25] := 2.0;
   DATA[2633,26] := 7.873815;
   DATA[2633,27] := 144.4758;
   DATA[2633,28] := 261.3753;
   DATA[2633,29] := 12.03538;
   DATA[2633,30] := 1.729428;
   DATA[2633,31] := 1.287691;
   DATA[2633,32] := 0.7352687;
   DATA[2633,33] := 0.3083624;
   DATA[2633,34] := 2.0;
   DATA[2633,35] := 250.4326;
   DATA[2633,36] := 1.746067;
   DATA[2633,37] := 189.1823;
   DATA[2633,38] := 0.000128152;
   DATA[2633,39] := 1.0;
   DATA[2633,40] := 1.0;
   DATA[2634,0] := 2.564135;
   DATA[2634,1] := 869.0168;
   DATA[2634,2] := 2.0;
   DATA[2634,3] := 2.0;
   DATA[2634,4] := 262.3366;
   DATA[2634,5] := 8.39868;
   DATA[2634,6] := 329.2745;
   DATA[2634,7] := 2.456156;
   DATA[2634,8] := 2.0;
   DATA[2634,9] := 2.0;
   DATA[2634,10] := 2.0;
   DATA[2634,11] := 19.71957;
   DATA[2634,12] := 2.206707;
   DATA[2634,13] := 832.0783;
   DATA[2634,14] := 1.0;
   DATA[2634,15] := 2.0;
   DATA[2634,16] := 1.0;
   DATA[2634,17] := 1.0;
   DATA[2634,18] := 1.0;
   DATA[2634,19] := 2.0;
   DATA[2634,20] := 148.808;
   DATA[2634,21] := 155.5499;
   DATA[2634,22] := 1.722359;
   DATA[2634,23] := 878.6208;
   DATA[2634,24] := 2.0;
   DATA[2634,25] := 2.0;
   DATA[2634,26] := 7.873815;
   DATA[2634,27] := 144.4758;
   DATA[2634,28] := 261.3753;
   DATA[2634,29] := 12.03538;
   DATA[2634,30] := 1.730582;
   DATA[2634,31] := 1.287434;
   DATA[2634,32] := 0.7352687;
   DATA[2634,33] := 0.3083624;
   DATA[2634,34] := 2.0;
   DATA[2634,35] := 250.4326;
   DATA[2634,36] := 1.746067;
   DATA[2634,37] := 189.1823;
   DATA[2634,38] := 0.000128152;
   DATA[2634,39] := 1.0;
   DATA[2634,40] := 1.0;
   DATA[2635,0] := 2.537232;
   DATA[2635,1] := 869.0561;
   DATA[2635,2] := 2.0;
   DATA[2635,3] := 2.0;
   DATA[2635,4] := 262.3366;
   DATA[2635,5] := 8.39868;
   DATA[2635,6] := 329.2745;
   DATA[2635,7] := 2.454234;
   DATA[2635,8] := 2.0;
   DATA[2635,9] := 2.0;
   DATA[2635,10] := 2.0;
   DATA[2635,11] := 19.72598;
   DATA[2635,12] := 2.206707;
   DATA[2635,13] := 831.9982;
   DATA[2635,14] := 1.0;
   DATA[2635,15] := 2.0;
   DATA[2635,16] := 1.0;
   DATA[2635,17] := 1.0;
   DATA[2635,18] := 1.0;
   DATA[2635,19] := 2.0;
   DATA[2635,20] := 148.808;
   DATA[2635,21] := 155.5499;
   DATA[2635,22] := 1.718771;
   DATA[2635,23] := 878.6208;
   DATA[2635,24] := 2.0;
   DATA[2635,25] := 2.0;
   DATA[2635,26] := 7.873815;
   DATA[2635,27] := 144.4758;
   DATA[2635,28] := 261.3753;
   DATA[2635,29] := 12.11228;
   DATA[2635,30] := 1.730582;
   DATA[2635,31] := 1.294479;
   DATA[2635,32] := 0.7352687;
   DATA[2635,33] := 0.3083624;
   DATA[2635,34] := 2.0;
   DATA[2635,35] := 250.2403;
   DATA[2635,36] := 1.665972;
   DATA[2635,37] := 188.958;
   DATA[2635,38] := 0.000128152;
   DATA[2635,39] := 1.0;
   DATA[2635,40] := 1.0;
   DATA[2636,0] := 2.517695;
   DATA[2636,1] := 869.2523;
   DATA[2636,2] := 2.0;
   DATA[2636,3] := 2.0;
   DATA[2636,4] := 262.3366;
   DATA[2636,5] := 8.39868;
   DATA[2636,6] := 329.2745;
   DATA[2636,7] := 2.454234;
   DATA[2636,8] := 2.0;
   DATA[2636,9] := 2.0;
   DATA[2636,10] := 2.0;
   DATA[2636,11] := 19.72598;
   DATA[2636,12] := 2.207475;
   DATA[2636,13] := 831.9982;
   DATA[2636,14] := 1.0;
   DATA[2636,15] := 2.0;
   DATA[2636,16] := 1.0;
   DATA[2636,17] := 1.0;
   DATA[2636,18] := 1.0;
   DATA[2636,19] := 2.0;
   DATA[2636,20] := 148.808;
   DATA[2636,21] := 155.5499;
   DATA[2636,22] := 1.717233;
   DATA[2636,23] := 878.467;
   DATA[2636,24] := 2.0;
   DATA[2636,25] := 2.0;
   DATA[2636,26] := 7.873815;
   DATA[2636,27] := 144.4758;
   DATA[2636,28] := 261.3753;
   DATA[2636,29] := 12.11228;
   DATA[2636,30] := 1.728531;
   DATA[2636,31] := 1.295632;
   DATA[2636,32] := 0.7352687;
   DATA[2636,33] := 0.3083624;
   DATA[2636,34] := 2.0;
   DATA[2636,35] := 250.1923;
   DATA[2636,36] := 1.665972;
   DATA[2636,37] := 188.958;
   DATA[2636,38] := 0.000128152;
   DATA[2636,39] := 1.0;
   DATA[2636,40] := 1.0;
   DATA[2637,0] := 2.498479;
   DATA[2637,1] := 869.3308;
   DATA[2637,2] := 2.0;
   DATA[2637,3] := 2.0;
   DATA[2637,4] := 262.3366;
   DATA[2637,5] := 8.39868;
   DATA[2637,6] := 329.2745;
   DATA[2637,7] := 2.454234;
   DATA[2637,8] := 2.0;
   DATA[2637,9] := 2.0;
   DATA[2637,10] := 2.0;
   DATA[2637,11] := 19.72598;
   DATA[2637,12] := 2.209397;
   DATA[2637,13] := 832.1985;
   DATA[2637,14] := 1.0;
   DATA[2637,15] := 2.0;
   DATA[2637,16] := 1.0;
   DATA[2637,17] := 1.0;
   DATA[2637,18] := 1.0;
   DATA[2637,19] := 2.0;
   DATA[2637,20] := 148.808;
   DATA[2637,21] := 155.5499;
   DATA[2637,22] := 1.715824;
   DATA[2637,23] := 878.5824;
   DATA[2637,24] := 2.0;
   DATA[2637,25] := 2.0;
   DATA[2637,26] := 7.873815;
   DATA[2637,27] := 144.4758;
   DATA[2637,28] := 261.3753;
   DATA[2637,29] := 12.11228;
   DATA[2637,30] := 1.728531;
   DATA[2637,31] := 1.30652;
   DATA[2637,32] := 0.7352687;
   DATA[2637,33] := 0.3083624;
   DATA[2637,34] := 2.0;
   DATA[2637,35] := 249.984;
   DATA[2637,36] := 1.665972;
   DATA[2637,37] := 188.958;
   DATA[2637,38] := 0.000128152;
   DATA[2637,39] := 1.0;
   DATA[2637,40] := 1.0;
   DATA[2638,0] := 2.477981;
   DATA[2638,1] := 869.8019;
   DATA[2638,2] := 2.0;
   DATA[2638,3] := 2.0;
   DATA[2638,4] := 262.3366;
   DATA[2638,5] := 8.39868;
   DATA[2638,6] := 329.2745;
   DATA[2638,7] := 2.454234;
   DATA[2638,8] := 2.0;
   DATA[2638,9] := 2.0;
   DATA[2638,10] := 2.0;
   DATA[2638,11] := 19.75159;
   DATA[2638,12] := 2.209397;
   DATA[2638,13] := 832.0783;
   DATA[2638,14] := 1.0;
   DATA[2638,15] := 2.0;
   DATA[2638,16] := 1.0;
   DATA[2638,17] := 1.0;
   DATA[2638,18] := 1.0;
   DATA[2638,19] := 2.0;
   DATA[2638,20] := 148.808;
   DATA[2638,21] := 155.5499;
   DATA[2638,22] := 1.714798;
   DATA[2638,23] := 878.8131;
   DATA[2638,24] := 2.0;
   DATA[2638,25] := 2.0;
   DATA[2638,26] := 7.873815;
   DATA[2638,27] := 144.4758;
   DATA[2638,28] := 261.3753;
   DATA[2638,29] := 12.11228;
   DATA[2638,30] := 1.728531;
   DATA[2638,31] := 1.302933;
   DATA[2638,32] := 0.7352687;
   DATA[2638,33] := 0.3083624;
   DATA[2638,34] := 2.0;
   DATA[2638,35] := 249.984;
   DATA[2638,36] := 1.665972;
   DATA[2638,37] := 188.8779;
   DATA[2638,38] := 0.000128152;
   DATA[2638,39] := 1.0;
   DATA[2638,40] := 1.0;
   DATA[2639,0] := 2.458444;
   DATA[2639,1] := 869.6448;
   DATA[2639,2] := 2.0;
   DATA[2639,3] := 2.0;
   DATA[2639,4] := 262.3366;
   DATA[2639,5] := 8.39868;
   DATA[2639,6] := 329.2745;
   DATA[2639,7] := 2.454234;
   DATA[2639,8] := 2.0;
   DATA[2639,9] := 2.0;
   DATA[2639,10] := 2.0;
   DATA[2639,11] := 19.65875;
   DATA[2639,12] := 2.209397;
   DATA[2639,13] := 832.2385;
   DATA[2639,14] := 1.0;
   DATA[2639,15] := 2.0;
   DATA[2639,16] := 1.0;
   DATA[2639,17] := 1.0;
   DATA[2639,18] := 1.0;
   DATA[2639,19] := 2.0;
   DATA[2639,20] := 148.808;
   DATA[2639,21] := 155.5499;
   DATA[2639,22] := 1.714542;
   DATA[2639,23] := 879.3514;
   DATA[2639,24] := 2.0;
   DATA[2639,25] := 2.0;
   DATA[2639,26] := 7.873815;
   DATA[2639,27] := 144.5783;
   DATA[2639,28] := 261.3753;
   DATA[2639,29] := 12.11228;
   DATA[2639,30] := 1.728531;
   DATA[2639,31] := 1.285129;
   DATA[2639,32] := 0.7352687;
   DATA[2639,33] := 0.3083624;
   DATA[2639,34] := 2.0;
   DATA[2639,35] := 249.984;
   DATA[2639,36] := 1.665972;
   DATA[2639,37] := 188.8618;
   DATA[2639,38] := 0.000128152;
   DATA[2639,39] := 1.0;
   DATA[2639,40] := 1.0;
   DATA[2640,0] := 2.444031;
   DATA[2640,1] := 869.4486;
   DATA[2640,2] := 2.0;
   DATA[2640,3] := 2.0;
   DATA[2640,4] := 262.3366;
   DATA[2640,5] := 8.395475;
   DATA[2640,6] := 329.2745;
   DATA[2640,7] := 2.454234;
   DATA[2640,8] := 2.0;
   DATA[2640,9] := 2.0;
   DATA[2640,10] := 2.0;
   DATA[2640,11] := 19.65555;
   DATA[2640,12] := 2.209397;
   DATA[2640,13] := 832.0383;
   DATA[2640,14] := 1.0;
   DATA[2640,15] := 2.0;
   DATA[2640,16] := 1.0;
   DATA[2640,17] := 1.0;
   DATA[2640,18] := 1.0;
   DATA[2640,19] := 2.0;
   DATA[2640,20] := 148.808;
   DATA[2640,21] := 155.5499;
   DATA[2640,22] := 1.712363;
   DATA[2640,23] := 879.1976;
   DATA[2640,24] := 2.0;
   DATA[2640,25] := 2.0;
   DATA[2640,26] := 7.873815;
   DATA[2640,27] := 144.5783;
   DATA[2640,28] := 261.3753;
   DATA[2640,29] := 12.11228;
   DATA[2640,30] := 1.726993;
   DATA[2640,31] := 1.272704;
   DATA[2640,32] := 0.7352687;
   DATA[2640,33] := 0.3083624;
   DATA[2640,34] := 2.0;
   DATA[2640,35] := 249.984;
   DATA[2640,36] := 1.665972;
   DATA[2640,37] := 188.8618;
   DATA[2640,38] := 0.000128152;
   DATA[2640,39] := 1.0;
   DATA[2640,40] := 1.0;
   DATA[2641,0] := 2.426416;
   DATA[2641,1] := 869.6841;
   DATA[2641,2] := 2.0;
   DATA[2641,3] := 2.0;
   DATA[2641,4] := 262.3366;
   DATA[2641,5] := 8.395475;
   DATA[2641,6] := 329.2745;
   DATA[2641,7] := 2.454234;
   DATA[2641,8] := 2.0;
   DATA[2641,9] := 2.0;
   DATA[2641,10] := 2.0;
   DATA[2641,11] := 19.65555;
   DATA[2641,12] := 2.209397;
   DATA[2641,13] := 831.838;
   DATA[2641,14] := 1.0;
   DATA[2641,15] := 2.0;
   DATA[2641,16] := 1.0;
   DATA[2641,17] := 1.0;
   DATA[2641,18] := 1.0;
   DATA[2641,19] := 2.0;
   DATA[2641,20] := 148.808;
   DATA[2641,21] := 155.4217;
   DATA[2641,22] := 1.712363;
   DATA[2641,23] := 879.3514;
   DATA[2641,24] := 2.0;
   DATA[2641,25] := 2.0;
   DATA[2641,26] := 7.873815;
   DATA[2641,27] := 144.5783;
   DATA[2641,28] := 261.3753;
   DATA[2641,29] := 12.11228;
   DATA[2641,30] := 1.725968;
   DATA[2641,31] := 1.277187;
   DATA[2641,32] := 0.7352687;
   DATA[2641,33] := 0.3083624;
   DATA[2641,34] := 2.0;
   DATA[2641,35] := 249.984;
   DATA[2641,36] := 1.665972;
   DATA[2641,37] := 188.8618;
   DATA[2641,38] := 0.000128152;
   DATA[2641,39] := 1.0;
   DATA[2641,40] := 1.0;
   DATA[2642,0] := 2.421612;
   DATA[2642,1] := 869.5271;
   DATA[2642,2] := 2.0;
   DATA[2642,3] := 2.0;
   DATA[2642,4] := 262.3366;
   DATA[2642,5] := 8.395475;
   DATA[2642,6] := 329.2745;
   DATA[2642,7] := 2.454234;
   DATA[2642,8] := 2.0;
   DATA[2642,9] := 2.0;
   DATA[2642,10] := 2.0;
   DATA[2642,11] := 19.65555;
   DATA[2642,12] := 2.209397;
   DATA[2642,13] := 832.0783;
   DATA[2642,14] := 1.0;
   DATA[2642,15] := 2.0;
   DATA[2642,16] := 1.0;
   DATA[2642,17] := 1.0;
   DATA[2642,18] := 1.0;
   DATA[2642,19] := 2.0;
   DATA[2642,20] := 148.808;
   DATA[2642,21] := 155.3192;
   DATA[2642,22] := 1.713645;
   DATA[2642,23] := 879.8129;
   DATA[2642,24] := 2.0;
   DATA[2642,25] := 2.0;
   DATA[2642,26] := 7.873815;
   DATA[2642,27] := 144.5783;
   DATA[2642,28] := 261.3753;
   DATA[2642,29] := 12.11228;
   DATA[2642,30] := 1.725968;
   DATA[2642,31] := 1.281158;
   DATA[2642,32] := 0.7352687;
   DATA[2642,33] := 0.3083624;
   DATA[2642,34] := 2.0;
   DATA[2642,35] := 249.984;
   DATA[2642,36] := 1.665972;
   DATA[2642,37] := 188.8618;
   DATA[2642,38] := 0.000128152;
   DATA[2642,39] := 1.0;
   DATA[2642,40] := 1.0;
   DATA[2643,0] := 2.424815;
   DATA[2643,1] := 869.6056;
   DATA[2643,2] := 2.0;
   DATA[2643,3] := 2.0;
   DATA[2643,4] := 262.3366;
   DATA[2643,5] := 8.393873;
   DATA[2643,6] := 329.2745;
   DATA[2643,7] := 2.454234;
   DATA[2643,8] := 2.0;
   DATA[2643,9] := 2.0;
   DATA[2643,10] := 2.0;
   DATA[2643,11] := 19.69076;
   DATA[2643,12] := 2.209397;
   DATA[2643,13] := 832.3587;
   DATA[2643,14] := 1.0;
   DATA[2643,15] := 2.0;
   DATA[2643,16] := 1.0;
   DATA[2643,17] := 1.0;
   DATA[2643,18] := 1.0;
   DATA[2643,19] := 2.0;
   DATA[2643,20] := 148.808;
   DATA[2643,21] := 155.3192;
   DATA[2643,22] := 1.714798;
   DATA[2643,23] := 879.9667;
   DATA[2643,24] := 2.0;
   DATA[2643,25] := 2.0;
   DATA[2643,26] := 7.873815;
   DATA[2643,27] := 144.7578;
   DATA[2643,28] := 261.3753;
   DATA[2643,29] := 12.11228;
   DATA[2643,30] := 1.725455;
   DATA[2643,31] := 1.29243;
   DATA[2643,32] := 0.7352687;
   DATA[2643,33] := 0.3083624;
   DATA[2643,34] := 2.0;
   DATA[2643,35] := 249.984;
   DATA[2643,36] := 1.665972;
   DATA[2643,37] := 188.8618;
   DATA[2643,38] := 0.000128152;
   DATA[2643,39] := 1.0;
   DATA[2643,40] := 1.0;
   DATA[2644,0] := 2.445633;
   DATA[2644,1] := 869.7234;
   DATA[2644,2] := 2.0;
   DATA[2644,3] := 2.0;
   DATA[2644,4] := 262.3366;
   DATA[2644,5] := 8.393873;
   DATA[2644,6] := 329.2745;
   DATA[2644,7] := 2.454362;
   DATA[2644,8] := 2.0;
   DATA[2644,9] := 2.0;
   DATA[2644,10] := 2.0;
   DATA[2644,11] := 19.69396;
   DATA[2644,12] := 2.209397;
   DATA[2644,13] := 832.7593;
   DATA[2644,14] := 1.0;
   DATA[2644,15] := 2.0;
   DATA[2644,16] := 1.0;
   DATA[2644,17] := 1.0;
   DATA[2644,18] := 1.0;
   DATA[2644,19] := 2.0;
   DATA[2644,20] := 148.808;
   DATA[2644,21] := 155.2935;
   DATA[2644,22] := 1.714798;
   DATA[2644,23] := 880.1205;
   DATA[2644,24] := 2.0;
   DATA[2644,25] := 2.0;
   DATA[2644,26] := 7.873815;
   DATA[2644,27] := 144.7578;
   DATA[2644,28] := 261.3753;
   DATA[2644,29] := 12.11228;
   DATA[2644,30] := 1.725455;
   DATA[2644,31] := 1.29243;
   DATA[2644,32] := 0.7352687;
   DATA[2644,33] := 0.3083624;
   DATA[2644,34] := 2.0;
   DATA[2644,35] := 250.2403;
   DATA[2644,36] := 1.665972;
   DATA[2644,37] := 188.8618;
   DATA[2644,38] := 0.000128152;
   DATA[2644,39] := 1.0;
   DATA[2644,40] := 1.0;
   DATA[2645,0] := 2.518656;
   DATA[2645,1] := 869.4486;
   DATA[2645,2] := 2.0;
   DATA[2645,3] := 2.0;
   DATA[2645,4] := 262.3366;
   DATA[2645,5] := 8.393873;
   DATA[2645,6] := 329.2745;
   DATA[2645,7] := 2.455131;
   DATA[2645,8] := 2.0;
   DATA[2645,9] := 2.0;
   DATA[2645,10] := 2.0;
   DATA[2645,11] := 19.69396;
   DATA[2645,12] := 2.209397;
   DATA[2645,13] := 833.36;
   DATA[2645,14] := 1.0;
   DATA[2645,15] := 2.0;
   DATA[2645,16] := 1.0;
   DATA[2645,17] := 1.0;
   DATA[2645,18] := 1.0;
   DATA[2645,19] := 2.0;
   DATA[2645,20] := 148.808;
   DATA[2645,21] := 155.191;
   DATA[2645,22] := 1.717105;
   DATA[2645,23] := 880.1589;
   DATA[2645,24] := 2.0;
   DATA[2645,25] := 2.0;
   DATA[2645,26] := 7.873815;
   DATA[2645,27] := 144.7578;
   DATA[2645,28] := 261.3753;
   DATA[2645,29] := 12.11228;
   DATA[2645,30] := 1.725455;
   DATA[2645,31] := 1.28705;
   DATA[2645,32] := 0.7352687;
   DATA[2645,33] := 0.3083624;
   DATA[2645,34] := 2.0;
   DATA[2645,35] := 250.2403;
   DATA[2645,36] := 1.665972;
   DATA[2645,37] := 188.9259;
   DATA[2645,38] := 0.000128152;
   DATA[2645,39] := 1.0;
   DATA[2645,40] := 1.0;
   DATA[2646,0] := 2.539474;
   DATA[2646,1] := 869.8804;
   DATA[2646,2] := 2.0;
   DATA[2646,3] := 2.0;
   DATA[2646,4] := 262.3366;
   DATA[2646,5] := 8.393873;
   DATA[2646,6] := 329.2745;
   DATA[2646,7] := 2.455131;
   DATA[2646,8] := 2.0;
   DATA[2646,9] := 2.0;
   DATA[2646,10] := 2.0;
   DATA[2646,11] := 19.69396;
   DATA[2646,12] := 2.209397;
   DATA[2646,13] := 833.5603;
   DATA[2646,14] := 1.0;
   DATA[2646,15] := 2.0;
   DATA[2646,16] := 1.0;
   DATA[2646,17] := 1.0;
   DATA[2646,18] := 1.0;
   DATA[2646,19] := 2.0;
   DATA[2646,20] := 148.808;
   DATA[2646,21] := 155.191;
   DATA[2646,22] := 1.717105;
   DATA[2646,23] := 880.3127;
   DATA[2646,24] := 2.0;
   DATA[2646,25] := 2.0;
   DATA[2646,26] := 7.873815;
   DATA[2646,27] := 144.7578;
   DATA[2646,28] := 261.3753;
   DATA[2646,29] := 12.07383;
   DATA[2646,30] := 1.725711;
   DATA[2646,31] := 1.28705;
   DATA[2646,32] := 0.7352687;
   DATA[2646,33] := 0.3066329;
   DATA[2646,34] := 2.0;
   DATA[2646,35] := 250.2403;
   DATA[2646,36] := 1.665972;
   DATA[2646,37] := 189.022;
   DATA[2646,38] := 0.000128152;
   DATA[2646,39] := 1.0;
   DATA[2646,40] := 1.0;
   DATA[2647,0] := 2.595202;
   DATA[2647,1] := 869.8411;
   DATA[2647,2] := 2.0;
   DATA[2647,3] := 2.0;
   DATA[2647,4] := 262.3366;
   DATA[2647,5] := 8.393873;
   DATA[2647,6] := 329.2745;
   DATA[2647,7] := 2.454362;
   DATA[2647,8] := 2.0;
   DATA[2647,9] := 2.0;
   DATA[2647,10] := 2.0;
   DATA[2647,11] := 19.69396;
   DATA[2647,12] := 2.209397;
   DATA[2647,13] := 833.4402;
   DATA[2647,14] := 1.0;
   DATA[2647,15] := 2.0;
   DATA[2647,16] := 1.0;
   DATA[2647,17] := 1.0;
   DATA[2647,18] := 1.0;
   DATA[2647,19] := 2.0;
   DATA[2647,20] := 148.808;
   DATA[2647,21] := 155.191;
   DATA[2647,22] := 1.718002;
   DATA[2647,23] := 880.8895;
   DATA[2647,24] := 2.0;
   DATA[2647,25] := 2.0;
   DATA[2647,26] := 7.873815;
   DATA[2647,27] := 144.7578;
   DATA[2647,28] := 261.3753;
   DATA[2647,29] := 12.03538;
   DATA[2647,30] := 1.726096;
   DATA[2647,31] := 1.281286;
   DATA[2647,32] := 0.7352687;
   DATA[2647,33] := 0.3065048;
   DATA[2647,34] := 2.0;
   DATA[2647,35] := 250.2403;
   DATA[2647,36] := 1.730048;
   DATA[2647,37] := 189.1182;
   DATA[2647,38] := 0.000128152;
   DATA[2647,39] := 1.0;
   DATA[2647,40] := 1.0;
   DATA[2648,0] := 2.620504;
   DATA[2648,1] := 869.4094;
   DATA[2648,2] := 2.0;
   DATA[2648,3] := 2.0;
   DATA[2648,4] := 262.3366;
   DATA[2648,5] := 8.393873;
   DATA[2648,6] := 329.2745;
   DATA[2648,7] := 2.45308;
   DATA[2648,8] := 2.0;
   DATA[2648,9] := 2.0;
   DATA[2648,10] := 2.0;
   DATA[2648,11] := 19.66835;
   DATA[2648,12] := 2.209397;
   DATA[2648,13] := 833.6404;
   DATA[2648,14] := 1.0;
   DATA[2648,15] := 2.0;
   DATA[2648,16] := 1.0;
   DATA[2648,17] := 1.0;
   DATA[2648,18] := 1.0;
   DATA[2648,19] := 2.0;
   DATA[2648,20] := 148.808;
   DATA[2648,21] := 155.191;
   DATA[2648,22] := 1.718387;
   DATA[2648,23] := 880.8895;
   DATA[2648,24] := 2.0;
   DATA[2648,25] := 2.0;
   DATA[2648,26] := 7.873815;
   DATA[2648,27] := 144.7578;
   DATA[2648,28] := 261.183;
   DATA[2648,29] := 12.03538;
   DATA[2648,30] := 1.726993;
   DATA[2648,31] := 1.28103;
   DATA[2648,32] := 0.7352687;
   DATA[2648,33] := 0.3065048;
   DATA[2648,34] := 2.0;
   DATA[2648,35] := 250.2403;
   DATA[2648,36] := 1.730048;
   DATA[2648,37] := 189.1182;
   DATA[2648,38] := 0.000128152;
   DATA[2648,39] := 1.0;
   DATA[2648,40] := 1.0;
   DATA[2649,0] := 2.656055;
   DATA[2649,1] := 869.4879;
   DATA[2649,2] := 2.0;
   DATA[2649,3] := 2.0;
   DATA[2649,4] := 262.3366;
   DATA[2649,5] := 8.393873;
   DATA[2649,6] := 329.2745;
   DATA[2649,7] := 2.45308;
   DATA[2649,8] := 2.0;
   DATA[2649,9] := 2.0;
   DATA[2649,10] := 2.0;
   DATA[2649,11] := 19.66835;
   DATA[2649,12] := 2.209397;
   DATA[2649,13] := 833.36;
   DATA[2649,14] := 1.0;
   DATA[2649,15] := 2.0;
   DATA[2649,16] := 1.0;
   DATA[2649,17] := 1.0;
   DATA[2649,18] := 1.0;
   DATA[2649,19] := 2.0;
   DATA[2649,20] := 148.808;
   DATA[2649,21] := 155.191;
   DATA[2649,22] := 1.720437;
   DATA[2649,23] := 881.1587;
   DATA[2649,24] := 2.0;
   DATA[2649,25] := 2.0;
   DATA[2649,26] := 7.874776;
   DATA[2649,27] := 144.7578;
   DATA[2649,28] := 261.183;
   DATA[2649,29] := 12.03538;
   DATA[2649,30] := 1.726993;
   DATA[2649,31] := 1.28103;
   DATA[2649,32] := 0.7352687;
   DATA[2649,33] := 0.3065048;
   DATA[2649,34] := 2.0;
   DATA[2649,35] := 250.2403;
   DATA[2649,36] := 1.730048;
   DATA[2649,37] := 189.1182;
   DATA[2649,38] := 0.000128152;
   DATA[2649,39] := 1.0;
   DATA[2649,40] := 1.0;
   DATA[2650,0] := 2.665663;
   DATA[2650,1] := 869.4094;
   DATA[2650,2] := 2.0;
   DATA[2650,3] := 2.0;
   DATA[2650,4] := 262.3366;
   DATA[2650,5] := 8.396757;
   DATA[2650,6] := 329.2745;
   DATA[2650,7] := 2.45308;
   DATA[2650,8] := 2.0;
   DATA[2650,9] := 2.0;
   DATA[2650,10] := 2.0;
   DATA[2650,11] := 19.74198;
   DATA[2650,12] := 2.209397;
   DATA[2650,13] := 833.36;
   DATA[2650,14] := 1.0;
   DATA[2650,15] := 2.0;
   DATA[2650,16] := 1.0;
   DATA[2650,17] := 1.0;
   DATA[2650,18] := 1.0;
   DATA[2650,19] := 2.0;
   DATA[2650,20] := 148.808;
   DATA[2650,21] := 155.191;
   DATA[2650,22] := 1.720437;
   DATA[2650,23] := 881.0433;
   DATA[2650,24] := 2.0;
   DATA[2650,25] := 2.0;
   DATA[2650,26] := 7.874776;
   DATA[2650,27] := 144.7578;
   DATA[2650,28] := 261.183;
   DATA[2650,29] := 12.03538;
   DATA[2650,30] := 1.727634;
   DATA[2650,31] := 1.273601;
   DATA[2650,32] := 0.7352687;
   DATA[2650,33] := 0.3065048;
   DATA[2650,34] := 2.0;
   DATA[2650,35] := 250.3525;
   DATA[2650,36] := 1.730048;
   DATA[2650,37] := 189.1182;
   DATA[2650,38] := 0.000128152;
   DATA[2650,39] := 1.0;
   DATA[2650,40] := 1.0;
   DATA[2651,0] := 2.665663;
   DATA[2651,1] := 869.5271;
   DATA[2651,2] := 2.0;
   DATA[2651,3] := 2.0;
   DATA[2651,4] := 262.3366;
   DATA[2651,5] := 8.396757;
   DATA[2651,6] := 329.1464;
   DATA[2651,7] := 2.454618;
   DATA[2651,8] := 2.0;
   DATA[2651,9] := 2.0;
   DATA[2651,10] := 2.0;
   DATA[2651,11] := 19.74198;
   DATA[2651,12] := 2.209397;
   DATA[2651,13] := 833.5603;
   DATA[2651,14] := 1.0;
   DATA[2651,15] := 2.0;
   DATA[2651,16] := 1.0;
   DATA[2651,17] := 1.0;
   DATA[2651,18] := 1.0;
   DATA[2651,19] := 2.0;
   DATA[2651,20] := 148.808;
   DATA[2651,21] := 155.191;
   DATA[2651,22] := 1.720437;
   DATA[2651,23] := 881.0433;
   DATA[2651,24] := 2.0;
   DATA[2651,25] := 2.0;
   DATA[2651,26] := 7.874776;
   DATA[2651,27] := 144.7578;
   DATA[2651,28] := 261.183;
   DATA[2651,29] := 12.03538;
   DATA[2651,30] := 1.728916;
   DATA[2651,31] := 1.277699;
   DATA[2651,32] := 0.7352687;
   DATA[2651,33] := 0.3065048;
   DATA[2651,34] := 2.0;
   DATA[2651,35] := 250.3525;
   DATA[2651,36] := 1.730048;
   DATA[2651,37] := 189.1182;
   DATA[2651,38] := 0.000128152;
   DATA[2651,39] := 1.0;
   DATA[2651,40] := 1.0;
   DATA[2652,0] := 2.65061;
   DATA[2652,1] := 869.8019;
   DATA[2652,2] := 2.0;
   DATA[2652,3] := 2.0;
   DATA[2652,4] := 262.3366;
   DATA[2652,5] := 8.396757;
   DATA[2652,6] := 329.1464;
   DATA[2652,7] := 2.454618;
   DATA[2652,8] := 2.0;
   DATA[2652,9] := 2.0;
   DATA[2652,10] := 2.0;
   DATA[2652,11] := 19.74198;
   DATA[2652,12] := 2.209397;
   DATA[2652,13] := 833.6004;
   DATA[2652,14] := 1.0;
   DATA[2652,15] := 2.0;
   DATA[2652,16] := 1.0;
   DATA[2652,17] := 1.0;
   DATA[2652,18] := 1.0;
   DATA[2652,19] := 2.0;
   DATA[2652,20] := 148.808;
   DATA[2652,21] := 155.191;
   DATA[2652,22] := 1.720437;
   DATA[2652,23] := 881.1202;
   DATA[2652,24] := 2.0;
   DATA[2652,25] := 2.0;
   DATA[2652,26] := 7.874776;
   DATA[2652,27] := 144.6039;
   DATA[2652,28] := 261.2151;
   DATA[2652,29] := 12.03538;
   DATA[2652,30] := 1.7293;
   DATA[2652,31] := 1.293711;
   DATA[2652,32] := 0.7352687;
   DATA[2652,33] := 0.3065048;
   DATA[2652,34] := 2.0;
   DATA[2652,35] := 250.3525;
   DATA[2652,36] := 1.730048;
   DATA[2652,37] := 189.1182;
   DATA[2652,38] := 0.000128152;
   DATA[2652,39] := 1.0;
   DATA[2652,40] := 1.0;
   DATA[2653,0] := 2.62755;
   DATA[2653,1] := 869.8019;
   DATA[2653,2] := 2.0;
   DATA[2653,3] := 2.0;
   DATA[2653,4] := 262.3366;
   DATA[2653,5] := 8.396757;
   DATA[2653,6] := 329.1464;
   DATA[2653,7] := 2.455515;
   DATA[2653,8] := 2.0;
   DATA[2653,9] := 2.0;
   DATA[2653,10] := 2.0;
   DATA[2653,11] := 19.67476;
   DATA[2653,12] := 2.209397;
   DATA[2653,13] := 833.4802;
   DATA[2653,14] := 1.0;
   DATA[2653,15] := 2.0;
   DATA[2653,16] := 1.0;
   DATA[2653,17] := 1.0;
   DATA[2653,18] := 1.0;
   DATA[2653,19] := 2.0;
   DATA[2653,20] := 148.808;
   DATA[2653,21] := 155.191;
   DATA[2653,22] := 1.720437;
   DATA[2653,23] := 880.8895;
   DATA[2653,24] := 2.0;
   DATA[2653,25] := 2.0;
   DATA[2653,26] := 7.874776;
   DATA[2653,27] := 144.6039;
   DATA[2653,28] := 261.3432;
   DATA[2653,29] := 12.03538;
   DATA[2653,30] := 1.7293;
   DATA[2653,31] := 1.297041;
   DATA[2653,32] := 0.7352687;
   DATA[2653,33] := 0.3065048;
   DATA[2653,34] := 2.0;
   DATA[2653,35] := 250.3525;
   DATA[2653,36] := 1.730048;
   DATA[2653,37] := 189.1182;
   DATA[2653,38] := 0.000128152;
   DATA[2653,39] := 1.0;
   DATA[2653,40] := 1.0;
   DATA[2654,0] := 2.622746;
   DATA[2654,1] := 869.8411;
   DATA[2654,2] := 2.0;
   DATA[2654,3] := 2.0;
   DATA[2654,4] := 262.3366;
   DATA[2654,5] := 8.396757;
   DATA[2654,6] := 329.1464;
   DATA[2654,7] := 2.455515;
   DATA[2654,8] := 2.0;
   DATA[2654,9] := 2.0;
   DATA[2654,10] := 2.0;
   DATA[2654,11] := 19.67476;
   DATA[2654,12] := 2.209397;
   DATA[2654,13] := 833.7606;
   DATA[2654,14] := 1.0;
   DATA[2654,15] := 2.0;
   DATA[2654,16] := 1.0;
   DATA[2654,17] := 1.0;
   DATA[2654,18] := 1.0;
   DATA[2654,19] := 2.0;
   DATA[2654,20] := 148.808;
   DATA[2654,21] := 155.191;
   DATA[2654,22] := 1.720437;
   DATA[2654,23] := 880.7357;
   DATA[2654,24] := 2.0;
   DATA[2654,25] := 2.0;
   DATA[2654,26] := 7.874776;
   DATA[2654,27] := 144.6039;
   DATA[2654,28] := 261.3432;
   DATA[2654,29] := 12.03538;
   DATA[2654,30] := 1.7293;
   DATA[2654,31] := 1.296401;
   DATA[2654,32] := 0.7352687;
   DATA[2654,33] := 0.3065689;
   DATA[2654,34] := 2.0;
   DATA[2654,35] := 250.3525;
   DATA[2654,36] := 1.730048;
   DATA[2654,37] := 189.1342;
   DATA[2654,38] := 0.000128152;
   DATA[2654,39] := 1.0;
   DATA[2654,40] := 1.0;
   DATA[2655,0] := 2.607693;
   DATA[2655,1] := 869.4094;
   DATA[2655,2] := 2.0;
   DATA[2655,3] := 2.0;
   DATA[2655,4] := 262.3366;
   DATA[2655,5] := 8.396757;
   DATA[2655,6] := 329.1464;
   DATA[2655,7] := 2.455515;
   DATA[2655,8] := 2.0;
   DATA[2655,9] := 2.0;
   DATA[2655,10] := 2.0;
   DATA[2655,11] := 19.62033;
   DATA[2655,12] := 2.209397;
   DATA[2655,13] := 833.6404;
   DATA[2655,14] := 1.0;
   DATA[2655,15] := 2.0;
   DATA[2655,16] := 1.0;
   DATA[2655,17] := 1.0;
   DATA[2655,18] := 1.0;
   DATA[2655,19] := 2.0;
   DATA[2655,20] := 148.808;
   DATA[2655,21] := 155.3961;
   DATA[2655,22] := 1.720437;
   DATA[2655,23] := 880.928;
   DATA[2655,24] := 2.0;
   DATA[2655,25] := 2.0;
   DATA[2655,26] := 7.874776;
   DATA[2655,27] := 144.6039;
   DATA[2655,28] := 261.3432;
   DATA[2655,29] := 12.03538;
   DATA[2655,30] := 1.7293;
   DATA[2655,31] := 1.296016;
   DATA[2655,32] := 0.7352687;
   DATA[2655,33] := 0.3066329;
   DATA[2655,34] := 2.0;
   DATA[2655,35] := 250.3525;
   DATA[2655,36] := 1.730048;
   DATA[2655,37] := 189.1662;
   DATA[2655,38] := 0.000128152;
   DATA[2655,39] := 1.0;
   DATA[2655,40] := 1.0;
   DATA[2656,0] := 2.587516;
   DATA[2656,1] := 869.8411;
   DATA[2656,2] := 2.0;
   DATA[2656,3] := 2.0;
   DATA[2656,4] := 262.3366;
   DATA[2656,5] := 8.396757;
   DATA[2656,6] := 329.1464;
   DATA[2656,7] := 2.455515;
   DATA[2656,8] := 2.0;
   DATA[2656,9] := 2.0;
   DATA[2656,10] := 2.0;
   DATA[2656,11] := 19.62033;
   DATA[2656,12] := 2.208884;
   DATA[2656,13] := 833.5603;
   DATA[2656,14] := 1.0;
   DATA[2656,15] := 2.0;
   DATA[2656,16] := 1.0;
   DATA[2656,17] := 1.0;
   DATA[2656,18] := 1.0;
   DATA[2656,19] := 2.0;
   DATA[2656,20] := 148.808;
   DATA[2656,21] := 155.3961;
   DATA[2656,22] := 1.720437;
   DATA[2656,23] := 880.7357;
   DATA[2656,24] := 2.0;
   DATA[2656,25] := 2.0;
   DATA[2656,26] := 7.874776;
   DATA[2656,27] := 144.6039;
   DATA[2656,28] := 261.3432;
   DATA[2656,29] := 12.03538;
   DATA[2656,30] := 1.7293;
   DATA[2656,31] := 1.292558;
   DATA[2656,32] := 0.7352687;
   DATA[2656,33] := 0.3066329;
   DATA[2656,34] := 2.0;
   DATA[2656,35] := 250.3525;
   DATA[2656,36] := 1.730048;
   DATA[2656,37] := 189.1662;
   DATA[2656,38] := 0.000128152;
   DATA[2656,39] := 1.0;
   DATA[2656,40] := 1.0;
   DATA[2657,0] := 2.562854;
   DATA[2657,1] := 870.0767;
   DATA[2657,2] := 2.0;
   DATA[2657,3] := 2.0;
   DATA[2657,4] := 262.3366;
   DATA[2657,5] := 8.396757;
   DATA[2657,6] := 329.1464;
   DATA[2657,7] := 2.455515;
   DATA[2657,8] := 2.0;
   DATA[2657,9] := 2.0;
   DATA[2657,10] := 2.0;
   DATA[2657,11] := 19.57232;
   DATA[2657,12] := 2.208884;
   DATA[2657,13] := 834.0009;
   DATA[2657,14] := 1.0;
   DATA[2657,15] := 2.0;
   DATA[2657,16] := 1.0;
   DATA[2657,17] := 1.0;
   DATA[2657,18] := 1.0;
   DATA[2657,19] := 2.0;
   DATA[2657,20] := 148.808;
   DATA[2657,21] := 155.3961;
   DATA[2657,22] := 1.720437;
   DATA[2657,23] := 880.4666;
   DATA[2657,24] := 2.0;
   DATA[2657,25] := 2.0;
   DATA[2657,26] := 7.873815;
   DATA[2657,27] := 144.6039;
   DATA[2657,28] := 261.3432;
   DATA[2657,29] := 12.03538;
   DATA[2657,30] := 1.7293;
   DATA[2657,31] := 1.291533;
   DATA[2657,32] := 0.7352687;
   DATA[2657,33] := 0.3066329;
   DATA[2657,34] := 2.0;
   DATA[2657,35] := 250.1762;
   DATA[2657,36] := 1.730048;
   DATA[2657,37] := 189.1662;
   DATA[2657,38] := 0.000128152;
   DATA[2657,39] := 1.0;
   DATA[2657,40] := 1.0;
   DATA[2658,0] := 2.537873;
   DATA[2658,1] := 869.7234;
   DATA[2658,2] := 2.0;
   DATA[2658,3] := 2.0;
   DATA[2658,4] := 262.3366;
   DATA[2658,5] := 8.396757;
   DATA[2658,6] := 329.1464;
   DATA[2658,7] := 2.452952;
   DATA[2658,8] := 2.0;
   DATA[2658,9] := 2.0;
   DATA[2658,10] := 2.0;
   DATA[2658,11] := 19.57232;
   DATA[2658,12] := 2.208884;
   DATA[2658,13] := 834.0009;
   DATA[2658,14] := 1.0;
   DATA[2658,15] := 2.0;
   DATA[2658,16] := 1.0;
   DATA[2658,17] := 1.0;
   DATA[2658,18] := 1.0;
   DATA[2658,19] := 2.0;
   DATA[2658,20] := 148.808;
   DATA[2658,21] := 155.3961;
   DATA[2658,22] := 1.720437;
   DATA[2658,23] := 880.8511;
   DATA[2658,24] := 2.0;
   DATA[2658,25] := 2.0;
   DATA[2658,26] := 7.873815;
   DATA[2658,27] := 144.6039;
   DATA[2658,28] := 261.3432;
   DATA[2658,29] := 12.03538;
   DATA[2658,30] := 1.7293;
   DATA[2658,31] := 1.291533;
   DATA[2658,32] := 0.7352687;
   DATA[2658,33] := 0.3066329;
   DATA[2658,34] := 2.0;
   DATA[2658,35] := 250.1762;
   DATA[2658,36] := 1.730048;
   DATA[2658,37] := 188.9419;
   DATA[2658,38] := 0.000128152;
   DATA[2658,39] := 1.0;
   DATA[2658,40] := 1.0;
   DATA[2659,0] := 2.521218;
   DATA[2659,1] := 869.8019;
   DATA[2659,2] := 2.0;
   DATA[2659,3] := 2.0;
   DATA[2659,4] := 262.3366;
   DATA[2659,5] := 8.396757;
   DATA[2659,6] := 329.1464;
   DATA[2659,7] := 2.452952;
   DATA[2659,8] := 2.0;
   DATA[2659,9] := 2.0;
   DATA[2659,10] := 2.0;
   DATA[2659,11] := 19.62674;
   DATA[2659,12] := 2.209653;
   DATA[2659,13] := 834.0009;
   DATA[2659,14] := 1.0;
   DATA[2659,15] := 2.0;
   DATA[2659,16] := 1.0;
   DATA[2659,17] := 1.0;
   DATA[2659,18] := 1.0;
   DATA[2659,19] := 2.0;
   DATA[2659,20] := 148.808;
   DATA[2659,21] := 155.3961;
   DATA[2659,22] := 1.718002;
   DATA[2659,23] := 880.6588;
   DATA[2659,24] := 2.0;
   DATA[2659,25] := 2.0;
   DATA[2659,26] := 7.872853;
   DATA[2659,27] := 144.6039;
   DATA[2659,28] := 261.3432;
   DATA[2659,29] := 12.03538;
   DATA[2659,30] := 1.7293;
   DATA[2659,31] := 1.291533;
   DATA[2659,32] := 0.7352687;
   DATA[2659,33] := 0.3066329;
   DATA[2659,34] := 2.0;
   DATA[2659,35] := 249.9519;
   DATA[2659,36] := 1.730048;
   DATA[2659,37] := 188.8618;
   DATA[2659,38] := 0.000128152;
   DATA[2659,39] := 1.0;
   DATA[2659,40] := 1.0;
   DATA[2660,0] := 2.500721;
   DATA[2660,1] := 869.9196;
   DATA[2660,2] := 2.0;
   DATA[2660,3] := 2.0;
   DATA[2660,4] := 262.3366;
   DATA[2660,5] := 8.396757;
   DATA[2660,6] := 329.1464;
   DATA[2660,7] := 2.452952;
   DATA[2660,8] := 2.0;
   DATA[2660,9] := 2.0;
   DATA[2660,10] := 2.0;
   DATA[2660,11] := 19.62674;
   DATA[2660,12] := 2.209653;
   DATA[2660,13] := 834.1611;
   DATA[2660,14] := 1.0;
   DATA[2660,15] := 2.0;
   DATA[2660,16] := 1.0;
   DATA[2660,17] := 1.0;
   DATA[2660,18] := 1.0;
   DATA[2660,19] := 2.0;
   DATA[2660,20] := 148.808;
   DATA[2660,21] := 155.3961;
   DATA[2660,22] := 1.717361;
   DATA[2660,23] := 881.0818;
   DATA[2660,24] := 2.0;
   DATA[2660,25] := 2.0;
   DATA[2660,26] := 7.872853;
   DATA[2660,27] := 144.6039;
   DATA[2660,28] := 261.3432;
   DATA[2660,29] := 12.03538;
   DATA[2660,30] := 1.7293;
   DATA[2660,31] := 1.28436;
   DATA[2660,32] := 0.7352687;
   DATA[2660,33] := 0.3066329;
   DATA[2660,34] := 2.0;
   DATA[2660,35] := 249.9519;
   DATA[2660,36] := 1.730048;
   DATA[2660,37] := 188.8618;
   DATA[2660,38] := 0.000128152;
   DATA[2660,39] := 1.0;
   DATA[2660,40] := 1.0;
   DATA[2661,0] := 2.483426;
   DATA[2661,1] := 870.1159;
   DATA[2661,2] := 2.0;
   DATA[2661,3] := 2.0;
   DATA[2661,4] := 262.3366;
   DATA[2661,5] := 8.396757;
   DATA[2661,6] := 329.1464;
   DATA[2661,7] := 2.452952;
   DATA[2661,8] := 2.0;
   DATA[2661,9] := 2.0;
   DATA[2661,10] := 2.0;
   DATA[2661,11] := 19.62674;
   DATA[2661,12] := 2.209653;
   DATA[2661,13] := 833.6004;
   DATA[2661,14] := 1.0;
   DATA[2661,15] := 2.0;
   DATA[2661,16] := 1.0;
   DATA[2661,17] := 1.0;
   DATA[2661,18] := 1.0;
   DATA[2661,19] := 2.0;
   DATA[2661,20] := 148.808;
   DATA[2661,21] := 155.3961;
   DATA[2661,22] := 1.717233;
   DATA[2661,23] := 880.7742;
   DATA[2661,24] := 2.0;
   DATA[2661,25] := 2.0;
   DATA[2661,26] := 7.872853;
   DATA[2661,27] := 144.7065;
   DATA[2661,28] := 261.3432;
   DATA[2661,29] := 12.03538;
   DATA[2661,30] := 1.7293;
   DATA[2661,31] := 1.286922;
   DATA[2661,32] := 0.7352687;
   DATA[2661,33] := 0.3066329;
   DATA[2661,34] := 2.0;
   DATA[2661,35] := 249.9519;
   DATA[2661,36] := 1.730048;
   DATA[2661,37] := 188.8618;
   DATA[2661,38] := 0.000128152;
   DATA[2661,39] := 1.0;
   DATA[2661,40] := 1.0;
   DATA[2662,0] := 2.468052;
   DATA[2662,1] := 870.2729;
   DATA[2662,2] := 2.0;
   DATA[2662,3] := 2.0;
   DATA[2662,4] := 262.3366;
   DATA[2662,5] := 8.396757;
   DATA[2662,6] := 329.1464;
   DATA[2662,7] := 2.452952;
   DATA[2662,8] := 2.0;
   DATA[2662,9] := 2.0;
   DATA[2662,10] := 2.0;
   DATA[2662,11] := 19.67476;
   DATA[2662,12] := 2.208756;
   DATA[2662,13] := 833.5603;
   DATA[2662,14] := 1.0;
   DATA[2662,15] := 2.0;
   DATA[2662,16] := 1.0;
   DATA[2662,17] := 1.0;
   DATA[2662,18] := 1.0;
   DATA[2662,19] := 2.0;
   DATA[2662,20] := 148.808;
   DATA[2662,21] := 155.3961;
   DATA[2662,22] := 1.717233;
   DATA[2662,23] := 880.5819;
   DATA[2662,24] := 2.0;
   DATA[2662,25] := 2.0;
   DATA[2662,26] := 7.872853;
   DATA[2662,27] := 144.7065;
   DATA[2662,28] := 261.3432;
   DATA[2662,29] := 12.03538;
   DATA[2662,30] := 1.7293;
   DATA[2662,31] := 1.301012;
   DATA[2662,32] := 0.7352687;
   DATA[2662,33] := 0.3066329;
   DATA[2662,34] := 2.0;
   DATA[2662,35] := 249.9519;
   DATA[2662,36] := 1.730048;
   DATA[2662,37] := 188.8618;
   DATA[2662,38] := 0.000128152;
   DATA[2662,39] := 1.0;
   DATA[2662,40] := 1.0;
   DATA[2663,0] := 2.449156;
   DATA[2663,1] := 870.5084;
   DATA[2663,2] := 2.0;
   DATA[2663,3] := 2.0;
   DATA[2663,4] := 262.3366;
   DATA[2663,5] := 8.396757;
   DATA[2663,6] := 329.1464;
   DATA[2663,7] := 2.452952;
   DATA[2663,8] := 2.0;
   DATA[2663,9] := 2.0;
   DATA[2663,10] := 2.0;
   DATA[2663,11] := 19.69396;
   DATA[2663,12] := 2.208756;
   DATA[2663,13] := 833.8007;
   DATA[2663,14] := 1.0;
   DATA[2663,15] := 2.0;
   DATA[2663,16] := 1.0;
   DATA[2663,17] := 1.0;
   DATA[2663,18] := 1.0;
   DATA[2663,19] := 2.0;
   DATA[2663,20] := 148.808;
   DATA[2663,21] := 155.3961;
   DATA[2663,22] := 1.717233;
   DATA[2663,23] := 880.6973;
   DATA[2663,24] := 2.0;
   DATA[2663,25] := 2.0;
   DATA[2663,26] := 7.872853;
   DATA[2663,27] := 144.7065;
   DATA[2663,28] := 261.3432;
   DATA[2663,29] := 12.03538;
   DATA[2663,30] := 1.7293;
   DATA[2663,31] := 1.296529;
   DATA[2663,32] := 0.7352687;
   DATA[2663,33] := 0.3066329;
   DATA[2663,34] := 2.0;
   DATA[2663,35] := 249.9519;
   DATA[2663,36] := 1.730048;
   DATA[2663,37] := 188.8618;
   DATA[2663,38] := 0.000128152;
   DATA[2663,39] := 1.0;
   DATA[2663,40] := 1.0;
   DATA[2664,0] := 2.436665;
   DATA[2664,1] := 870.4299;
   DATA[2664,2] := 2.0;
   DATA[2664,3] := 2.0;
   DATA[2664,4] := 262.3366;
   DATA[2664,5] := 8.396757;
   DATA[2664,6] := 329.1464;
   DATA[2664,7] := 2.452055;
   DATA[2664,8] := 2.0;
   DATA[2664,9] := 2.0;
   DATA[2664,10] := 2.0;
   DATA[2664,11] := 19.69396;
   DATA[2664,12] := 2.206322;
   DATA[2664,13] := 834.0009;
   DATA[2664,14] := 1.0;
   DATA[2664,15] := 2.0;
   DATA[2664,16] := 1.0;
   DATA[2664,17] := 1.0;
   DATA[2664,18] := 1.0;
   DATA[2664,19] := 2.0;
   DATA[2664,20] := 148.808;
   DATA[2664,21] := 155.3961;
   DATA[2664,22] := 1.717233;
   DATA[2664,23] := 880.7357;
   DATA[2664,24] := 2.0;
   DATA[2664,25] := 2.0;
   DATA[2664,26] := 7.872853;
   DATA[2664,27] := 144.7065;
   DATA[2664,28] := 261.3432;
   DATA[2664,29] := 12.03538;
   DATA[2664,30] := 1.726352;
   DATA[2664,31] := 1.3005;
   DATA[2664,32] := 0.7352687;
   DATA[2664,33] := 0.3066329;
   DATA[2664,34] := 2.0;
   DATA[2664,35] := 250.016;
